LIN {X 0,Y 203.825,Z 341.839,A -85,B 0,C 180,E1 -22082.308,E2 -22082.308} C_VEL
LIN {X 0,Y 207.128,Z 331.94,A -85,B 0,C 180,E1 -22084.047,E2 -22084.047} C_VEL
LIN {X 0,Y 210.227,Z 321.194,A -85,B 0,C 180,E1 -22085.512,E2 -22085.512} C_VEL
LIN {X 0,Y 213.25,Z 308.254,A -85,B 0,C 180,E1 -22086.828,E2 -22086.828} C_VEL
LIN {X 0,Y 215.405,Z 295.863,A -85,B 0,C 180,E1 -22087.718,E2 -22087.718} C_VEL
LIN {X 0,Y 216.743,Z 283.352,A -85,B 0,C 180,E1 -22088.313,E2 -22088.313} C_VEL
LIN {X 0,Y 218.908,Z 244.295,A -85,B 0,C 180,E1 -22089.519,E2 -22089.519} C_VEL
LIN {X 0,Y 217.298,Z 231.269,A -85,B 0,C 180,E1 -22090.465,E2 -22090.465} C_VEL
LIN {X 0,Y 211.83,Z 218.17,A -85,B 0,C 180,E1 -22092.439,E2 -22092.439} C_VEL
LIN {X 0,Y 205.925,Z 205.87,A -85,B 0,C 180,E1 -22094.682,E2 -22094.682} C_VEL
LIN {X 0,Y 200.117,Z 195.617,A -85,B 0,C 180,E1 -22097.023,E2 -22097.023} C_VEL
LIN {X 0,Y 197.007,Z 190.479,A -85,B 0,C 180,E1 -22098.363,E2 -22098.363} C_VEL
LIN {X 0,Y 193.844,Z 185.323,A -85,B 0,C 180,E1 -22099.808,E2 -22099.808} C_VEL
LIN {X 0,Y 190.334,Z 180.05,A -85,B 0,C 180,E1 -22101.501,E2 -22101.501} C_VEL
LIN {X 0,Y 187.044,Z 175.102,A -85,B 0,C 180,E1 -22103.213,E2 -22103.213} C_VEL
LIN {X 0,Y 186.738,Z 174.302,A -85,B 0,C 180,E1 -22103.647,E2 -22103.647} C_VEL
LIN {X 0,Y 185.574,Z 170.368,A -85,B 0,C 180,E1 -22107.043,E2 -22107.043} C_VEL
LIN {X 0,Y 185.551,Z 170.374,A -85,B 0,C 180,E1 -22110.596,E2 -22110.596} C_VEL
LIN {X 0,Y 185.584,Z 170.368,A -85,B 0,C 180,E1 -22115.382,E2 -22115.382} C_VEL
LIN {X 0,Y 185.629,Z 170.346,A -85,B 0,C 180,E1 -22121.18,E2 -22121.18} C_VEL
LIN {X 0,Y 185.7,Z 170.339,A -85,B 0,C 180,E1 -22126.875,E2 -22126.875} C_VEL
LIN {X 0,Y 185.972,Z 170.301,A -85,B 0,C 180,E1 -22131.306,E2 -22131.306} C_VEL
LIN {X 0,Y 186.159,Z 170.279,A -85,B 0,C 180,E1 -22137.837,E2 -22137.837} C_VEL
LIN {X 0,Y 186.378,Z 170.27,A -85,B 0,C 180,E1 -22140,E2 -22140} C_VEL
LIN {X 0,Y 185.881,Z 170.319,A -85,B 0,C 180,E1 -22144.337,E2 -22144.337} C_VEL
LIN {X 0,Y 185.977,Z 170.301,A -85,B 0,C 180,E1 -22148.694,E2 -22148.694} C_VEL
LIN {X 0,Y 185.716,Z 170.338,A -85,B 0,C 180,E1 -22153.124,E2 -22153.124} C_VEL
LIN {X 0,Y 185.655,Z 170.356,A -85,B 0,C 180,E1 -22157.629,E2 -22157.629} C_VEL
LIN {X 0,Y 185.558,Z 170.372,A -85,B 0,C 180,E1 -22162.257,E2 -22162.257} C_VEL
LIN {X 0,Y 185.582,Z 170.355,A -85,B 0,C 180,E1 -22164.646,E2 -22164.646} C_VEL
LIN {X 0,Y 185.549,Z 170.373,A -85,B 0,C 180,E1 -22170.753,E2 -22170.753} C_VEL
LIN {X 0,Y 185.54,Z 170.42,A -85,B 0,C 180,E1 -22171.468,E2 -22171.468} C_VEL
LIN {X 0,Y 186.279,Z 172.794,A -85,B 0,C 180,E1 -22171.967,E2 -22171.967} C_VEL
LIN {X 0,Y 188.238,Z 175.079,A -85,B 0,C 180,E1 -22172.981,E2 -22172.981} C_VEL
LIN {X 0,Y 189.453,Z 176.043,A -85,B 0,C 180,E1 -22173.559,E2 -22173.559} C_VEL
LIN {X 0,Y 191.363,Z 179.22,A -85,B 0,C 180,E1 -22174.539,E2 -22174.539} C_VEL
LIN {X 0,Y 193.288,Z 181.243,A -85,B 0,C 180,E1 -22175.415,E2 -22175.415} C_VEL
LIN {X 0,Y 195.933,Z 184.898,A -85,B 0,C 180,E1 -22176.614,E2 -22176.614} C_VEL
LIN {X 0,Y 202.478,Z 194.218,A -85,B 0,C 180,E1 -22179.344,E2 -22179.344} C_VEL
LIN {X 0,Y 209.512,Z 205.182,A -85,B 0,C 180,E1 -22181.991,E2 -22181.991} C_VEL
LIN {X 0,Y 216.8,Z 218.051,A -85,B 0,C 180,E1 -22184.505,E2 -22184.505} C_VEL
LIN {X 0,Y 219.958,Z 224.99,A -85,B 0,C 180,E1 -22185.571,E2 -22185.571} C_VEL
LIN {X 0,Y 217.34,Z 271.32,A -85,B 0,C 180,E1 -22187.032,E2 -22187.032} C_VEL
LIN {X 0,Y 215.752,Z 284.741,A -85,B 0,C 180,E1 -22187.789,E2 -22187.789} C_VEL
LIN {X 0,Y 213.587,Z 297.23,A -85,B 0,C 180,E1 -22188.844,E2 -22188.844} C_VEL
LIN {X 0,Y 211.086,Z 308.418,A -85,B 0,C 180,E1 -22190.152,E2 -22190.152} C_VEL
LIN {X 0,Y 207.862,Z 319.901,A -85,B 0,C 180,E1 -22191.898,E2 -22191.898} C_VEL
LIN {X 0,Y 204.36,Z 330.28,A -85,B 0,C 180,E1 -22193.917,E2 -22193.917} C_VEL
LIN {X 0,Y 201.13,Z 338.74,A -85,B 0,C 180,E1 -22196.006,E2 -22196.006} C_VEL
LIN {X 0,Y 197.303,Z 347.887,A -85,B 0,C 180,E1 -22198.908,E2 -22198.908} C_VEL
LIN {X 0,Y 193.98,Z 355.197,A -85,B 0,C 180,E1 -22201.899,E2 -22201.899} C_VEL
LIN {X 0,Y 190.993,Z 361.05,A -85,B 0,C 180,E1 -22204.964,E2 -22204.964} C_VEL
LIN {X 0,Y 188.559,Z 365.644,A -85,B 0,C 180,E1 -22208.115,E2 -22208.115} C_VEL
LIN {X 0,Y 187.195,Z 368.068,A -85,B 0,C 180,E1 -22210.25,E2 -22210.25} C_VEL
LIN {X 0,Y 186.035,Z 370.036,A -85,B 0,C 180,E1 -22212.407,E2 -22212.407} C_VEL
LIN {X 0,Y 185.054,Z 371.59,A -85,B 0,C 180,E1 -22214.581,E2 -22214.581} C_VEL
LIN {X 0,Y 184.363,Z 372.721,A -85,B 0,C 180,E1 -22216.776,E2 -22216.776} C_VEL
LIN {X 0,Y 183.555,Z 373.727,A -85,B 0,C 180,E1 -22221.188,E2 -22221.188} C_VEL
LIN {X 0,Y 183.398,Z 373.324,A -85,B 0,C 180,E1 -22225.107,E2 -22225.107} C_VEL
LIN {X 0,Y 183.418,Z 372.318,A -85,B 0,C 180,E1 -22227.802,E2 -22227.802} C_VEL
LIN {X 0,Y 183.588,Z 371.05,A -85,B 0,C 180,E1 -22229.998,E2 -22229.998} C_VEL
LIN {X 0,Y 184.097,Z 368.377,A -85,B 0,C 180,E1 -22233.281,E2 -22233.281} C_VEL
LIN {X 0,Y 185.006,Z 364.704,A -85,B 0,C 180,E1 -22236.542,E2 -22236.542} C_VEL
LIN {X 0,Y 186.412,Z 359.922,A -85,B 0,C 180,E1 -22239.766,E2 -22239.766} C_VEL
LIN {X 0,Y 188.216,Z 353.896,A -85,B 0,C 180,E1 -22242.944,E2 -22242.944} C_VEL
LIN {X 0,Y 190.668,Z 346.391,A -85,B 0,C 180,E1 -22246.046,E2 -22246.046} C_VEL
LIN {X 0,Y 192.991,Z 338.37,A -85,B 0,C 180,E1 -22248.697,E2 -22248.697} C_VEL
LIN {X 0,Y 195.744,Z 328.329,A -85,B 0,C 180,E1 -22251.315,E2 -22251.315} C_VEL
LIN {X 0,Y 198.322,Z 317.738,A -85,B 0,C 180,E1 -22253.493,E2 -22253.493} C_VEL
LIN {X 0,Y 200.493,Z 307.494,A -85,B 0,C 180,E1 -22255.15,E2 -22255.15} C_VEL
LIN {X 0,Y 202.556,Z 295.274,A -85,B 0,C 180,E1 -22256.67,E2 -22256.67} C_VEL
LIN {X 0,Y 204.199,Z 282.413,A -85,B 0,C 180,E1 -22257.823,E2 -22257.823} C_VEL
LIN {X 0,Y 205.326,Z 269.929,A -85,B 0,C 180,E1 -22258.561,E2 -22258.561} C_VEL
LIN {X 0,Y 207.959,Z 212.141,A -85,B 0,C 180,E1 -22260.481,E2 -22260.481} C_VEL
LIN {X 0,Y 202.776,Z 200.79,A -85,B 0,C 180,E1 -22261.935,E2 -22261.935} C_VEL
LIN {X 0,Y 196.04,Z 188.2,A -85,B 0,C 180,E1 -22263.885,E2 -22263.885} C_VEL
LIN {X 0,Y 189.509,Z 177.653,A -85,B 0,C 180,E1 -22265.882,E2 -22265.882} C_VEL
LIN {X 0,Y 187.666,Z 174.56,A -85,B 0,C 180,E1 -22266.486,E2 -22266.486} C_VEL
LIN {X 0,Y 185.986,Z 172.118,A -85,B 0,C 180,E1 -22267.034,E2 -22267.034} C_VEL
LIN {X 0,Y 185.541,Z 170.37,A -85,B 0,C 180,E1 -22267.302,E2 -22267.302} C_VEL
LIN {X 0,Y 185.48,Z 170.377,A -85,B 0,C 180,E1 -22270.727,E2 -22270.727} C_VEL
LIN {X 0,Y 185.455,Z 170.382,A -85,B 0,C 180,E1 -22276.053,E2 -22276.053} C_VEL
LIN {X 0,Y 185.463,Z 170.384,A -85,B 0,C 180,E1 -22279.893,E2 -22279.893} C_VEL
LIN {X 0,Y 185.501,Z 170.372,A -85,B 0,C 180,E1 -22282.709,E2 -22282.709} C_VEL
LIN {X 0,Y 185.536,Z 170.368,A -85,B 0,C 180,E1 -22287.973,E2 -22287.973} C_VEL
LIN {X 0,Y 185.574,Z 170.369,A -85,B 0,C 180,E1 -22290.575,E2 -22290.575} C_VEL
LIN {X 0,Y 185.573,Z 170.371,A -85,B 0,C 180,E1 -22295.38,E2 -22295.38} C_VEL
LIN {X 0,Y 185.625,Z 170.363,A -85,B 0,C 180,E1 -22301.17,E2 -22301.17} C_VEL
LIN {X 0,Y 185.659,Z 170.346,A -85,B 0,C 180,E1 -22304.634,E2 -22304.634} C_VEL
LIN {X 0,Y 185.88,Z 170.324,A -85,B 0,C 180,E1 -22309.419,E2 -22309.419} C_VEL
LIN {X 0,Y 185.919,Z 170.277,A -85,B 0,C 180,E1 -22313.488,E2 -22313.488} C_VEL
LIN {X 0,Y 186.165,Z 170.283,A -85,B 0,C 180,E1 -22317.836,E2 -22317.836} C_VEL
LIN {X 0,Y 186.369,Z 170.269,A -85,B 0,C 180,E1 -22320,E2 -22320} C_VEL
LIN {X 0,Y 185.874,Z 170.331,A -85,B 0,C 180,E1 -22324.337,E2 -22324.337} C_VEL
LIN {X 0,Y 185.963,Z 170.32,A -85,B 0,C 180,E1 -22328.695,E2 -22328.695} C_VEL
LIN {X 0,Y 185.707,Z 170.353,A -85,B 0,C 180,E1 -22333.124,E2 -22333.124} C_VEL
LIN {X 0,Y 185.647,Z 170.362,A -85,B 0,C 180,E1 -22337.629,E2 -22337.629} C_VEL
LIN {X 0,Y 185.565,Z 170.374,A -85,B 0,C 180,E1 -22342.255,E2 -22342.255} C_VEL
LIN {X 0,Y 185.551,Z 170.377,A -85,B 0,C 180,E1 -22347.034,E2 -22347.034} C_VEL
LIN {X 0,Y 185.57,Z 170.372,A -85,B 0,C 180,E1 -22349.495,E2 -22349.495} C_VEL
LIN {X 0,Y 185.492,Z 170.384,A -85,B 0,C 180,E1 -22354.633,E2 -22354.633} C_VEL
LIN {X 0,Y 185.499,Z 170.382,A -85,B 0,C 180,E1 -22357.315,E2 -22357.315} C_VEL
LIN {X 0,Y 185.465,Z 170.385,A -85,B 0,C 180,E1 -22360.726,E2 -22360.726} C_VEL
LIN {X 0,Y 185.477,Z 170.429,A -85,B 0,C 180,E1 -22364.321,E2 -22364.321} C_VEL
LIN {X 0,Y 187.116,Z 176.397,A -85,B 0,C 180,E1 -22367.854,E2 -22367.854} C_VEL
LIN {X 0,Y 189.501,Z 180.912,A -85,B 0,C 180,E1 -22368.662,E2 -22368.662} C_VEL
LIN {X 0,Y 196.299,Z 194.335,A -85,B 0,C 180,E1 -22370.837,E2 -22370.837} C_VEL
LIN {X 0,Y 202.806,Z 209.945,A -85,B 0,C 180,E1 -22372.848,E2 -22372.848} C_VEL
LIN {X 0,Y 204.31,Z 214.184,A -85,B 0,C 180,E1 -22373.315,E2 -22373.315} C_VEL
LIN {X 0,Y 206.787,Z 238.922,A -85,B 0,C 180,E1 -22374.783,E2 -22374.783} C_VEL
LIN {X 0,Y 206.092,Z 255.09,A -85,B 0,C 180,E1 -22375.314,E2 -22375.314} C_VEL
LIN {X 0,Y 205.375,Z 260.94,A -85,B 0,C 180,E1 -22375.412,E2 -22375.412} C_VEL
LIN {X 0,Y 199.61,Z 279.931,A -85,B 0,C 180,E1 -22375.151,E2 -22375.151} C_VEL
LIN {X 0,Y 198.569,Z 285.744,A -85,B 0,C 180,E1 -22375.294,E2 -22375.294} C_VEL
LIN {X 0,Y 197.257,Z 298.93,A -85,B 0,C 180,E1 -22376.098,E2 -22376.098} C_VEL
LIN {X 0,Y 195.306,Z 311.132,A -85,B 0,C 180,E1 -22377.182,E2 -22377.182} C_VEL
LIN {X 0,Y 192.849,Z 323.444,A -85,B 0,C 180,E1 -22378.717,E2 -22378.717} C_VEL
LIN {X 0,Y 190.011,Z 335.076,A -85,B 0,C 180,E1 -22380.657,E2 -22380.657} C_VEL
LIN {X 0,Y 187.159,Z 345.553,A -85,B 0,C 180,E1 -22382.918,E2 -22382.918} C_VEL
LIN {X 0,Y 184.582,Z 354.112,A -85,B 0,C 180,E1 -22385.242,E2 -22385.242} C_VEL
LIN {X 0,Y 182.176,Z 362.221,A -85,B 0,C 180,E1 -22387.993,E2 -22387.993} C_VEL
LIN {X 0,Y 180.295,Z 368.577,A -85,B 0,C 180,E1 -22390.653,E2 -22390.653} C_VEL
LIN {X 0,Y 178.425,Z 375.015,A -85,B 0,C 180,E1 -22393.997,E2 -22393.997} C_VEL
LIN {X 0,Y 177.084,Z 380.127,A -85,B 0,C 180,E1 -22397.394,E2 -22397.394} C_VEL
LIN {X 0,Y 176.4,Z 384.098,A -85,B 0,C 180,E1 -22400.832,E2 -22400.832} C_VEL
LIN {X 0,Y 176.152,Z 386.138,A -85,B 0,C 180,E1 -22403.128,E2 -22403.128} C_VEL
LIN {X 0,Y 176.124,Z 388.127,A -85,B 0,C 180,E1 -22406.022,E2 -22406.022} C_VEL
LIN {X 0,Y 176.323,Z 389.721,A -85,B 0,C 180,E1 -22410.002,E2 -22410.002} C_VEL
LIN {X 0,Y 176.089,Z 390.069,A -85,B 0,C 180,E1 -22413.806,E2 -22413.806} C_VEL
LIN {X 0,Y 176.111,Z 389.563,A -85,B 0,C 180,E1 -22416.878,E2 -22416.878} C_VEL
LIN {X 0,Y 176.388,Z 388.699,A -85,B 0,C 180,E1 -22419.173,E2 -22419.173} C_VEL
LIN {X 0,Y 177.614,Z 385.754,A -85,B 0,C 180,E1 -22423.736,E2 -22423.736} C_VEL
LIN {X 0,Y 179.276,Z 382.422,A -85,B 0,C 180,E1 -22427.1,E2 -22427.1} C_VEL
LIN {X 0,Y 181.534,Z 378.034,A -85,B 0,C 180,E1 -22430.393,E2 -22430.393} C_VEL
LIN {X 0,Y 184.257,Z 372.571,A -85,B 0,C 180,E1 -22433.551,E2 -22433.551} C_VEL
LIN {X 0,Y 187.585,Z 365.547,A -85,B 0,C 180,E1 -22436.719,E2 -22436.719} C_VEL
LIN {X 0,Y 190.915,Z 358.498,A -85,B 0,C 180,E1 -22439.195,E2 -22439.195} C_VEL
LIN {X 0,Y 194.621,Z 350.018,A -85,B 0,C 180,E1 -22441.577,E2 -22441.577} C_VEL
LIN {X 0,Y 198.704,Z 339.558,A -85,B 0,C 180,E1 -22443.855,E2 -22443.855} C_VEL
LIN {X 0,Y 202.628,Z 327.799,A -85,B 0,C 180,E1 -22445.826,E2 -22445.826} C_VEL
LIN {X 0,Y 205.941,Z 316.005,A -85,B 0,C 180,E1 -22447.284,E2 -22447.284} C_VEL
LIN {X 0,Y 208.653,Z 303.751,A -85,B 0,C 180,E1 -22448.393,E2 -22448.393} C_VEL
LIN {X 0,Y 210.672,Z 290.311,A -85,B 0,C 180,E1 -22449.258,E2 -22449.258} C_VEL
LIN {X 0,Y 211.914,Z 275.449,A -85,B 0,C 180,E1 -22449.81,E2 -22449.81} C_VEL
LIN {X 0,Y 213.594,Z 245.006,A -85,B 0,C 180,E1 -22450.76,E2 -22450.76} C_VEL
LIN {X 0,Y 212.13,Z 233.739,A -85,B 0,C 180,E1 -22451.641,E2 -22451.641} C_VEL
LIN {X 0,Y 206.753,Z 220.825,A -85,B 0,C 180,E1 -22453.705,E2 -22453.705} C_VEL
LIN {X 0,Y 201.579,Z 210.06,A -85,B 0,C 180,E1 -22455.79,E2 -22455.79} C_VEL
LIN {X 0,Y 196.244,Z 200.349,A -85,B 0,C 180,E1 -22458.077,E2 -22458.077} C_VEL
LIN {X 0,Y 192.932,Z 194.79,A -85,B 0,C 180,E1 -22459.594,E2 -22459.594} C_VEL
LIN {X 0,Y 190.321,Z 190.463,A -85,B 0,C 180,E1 -22460.862,E2 -22460.862} C_VEL
LIN {X 0,Y 187.146,Z 185.561,A -85,B 0,C 180,E1 -22462.484,E2 -22462.484} C_VEL
LIN {X 0,Y 183.366,Z 179.911,A -85,B 0,C 180,E1 -22464.57,E2 -22464.57} C_VEL
LIN {X 0,Y 180.11,Z 175.501,A -85,B 0,C 180,E1 -22466.505,E2 -22466.505} C_VEL
LIN {X 0,Y 179.416,Z 173.944,A -85,B 0,C 180,E1 -22467.078,E2 -22467.078} C_VEL
LIN {X 0,Y 178.465,Z 171.254,A -85,B 0,C 180,E1 -22469.876,E2 -22469.876} C_VEL
LIN {X 0,Y 178.519,Z 171.247,A -85,B 0,C 180,E1 -22474.89,E2 -22474.89} C_VEL
LIN {X 0,Y 178.609,Z 171.223,A -85,B 0,C 180,E1 -22481.652,E2 -22481.652} C_VEL
LIN {X 0,Y 178.627,Z 171.216,A -85,B 0,C 180,E1 -22486.346,E2 -22486.346} C_VEL
LIN {X 0,Y 178.904,Z 171.182,A -85,B 0,C 180,E1 -22490.96,E2 -22490.96} C_VEL
LIN {X 0,Y 178.819,Z 171.202,A -85,B 0,C 180,E1 -22495.492,E2 -22495.492} C_VEL
LIN {X 0,Y 179.343,Z 171.147,A -85,B 0,C 180,E1 -22500,E2 -22500} C_VEL
LIN {X 0,Y 178.831,Z 171.198,A -85,B 0,C 180,E1 -22504.508,E2 -22504.508} C_VEL
LIN {X 0,Y 178.908,Z 171.181,A -85,B 0,C 180,E1 -22509.041,E2 -22509.041} C_VEL
LIN {X 0,Y 178.642,Z 171.216,A -85,B 0,C 180,E1 -22513.654,E2 -22513.654} C_VEL
LIN {X 0,Y 178.558,Z 171.228,A -85,B 0,C 180,E1 -22519.151,E2 -22519.151} C_VEL
LIN {X 0,Y 178.52,Z 171.236,A -85,B 0,C 180,E1 -22525.111,E2 -22525.111} C_VEL
LIN {X 0,Y 178.461,Z 171.248,A -85,B 0,C 180,E1 -22527.962,E2 -22527.962} C_VEL
LIN {X 0,Y 179.101,Z 173.444,A -85,B 0,C 180,E1 -22528.481,E2 -22528.481} C_VEL
LIN {X 0,Y 181.05,Z 175.861,A -85,B 0,C 180,E1 -22529.68,E2 -22529.68} C_VEL
LIN {X 0,Y 182.667,Z 177.067,A -85,B 0,C 180,E1 -22530.57,E2 -22530.57} C_VEL
LIN {X 0,Y 184.522,Z 180.126,A -85,B 0,C 180,E1 -22531.662,E2 -22531.662} C_VEL
LIN {X 0,Y 186.707,Z 182.45,A -85,B 0,C 180,E1 -22532.798,E2 -22532.798} C_VEL
LIN {X 0,Y 189.354,Z 186.09,A -85,B 0,C 180,E1 -22534.151,E2 -22534.151} C_VEL
LIN {X 0,Y 190.879,Z 188.134,A -85,B 0,C 180,E1 -22534.892,E2 -22534.892} C_VEL
LIN {X 0,Y 194.087,Z 192.584,A -85,B 0,C 180,E1 -22536.382,E2 -22536.382} C_VEL
LIN {X 0,Y 199.121,Z 199.852,A -85,B 0,C 180,E1 -22538.551,E2 -22538.551} C_VEL
LIN {X 0,Y 205.658,Z 210.313,A -85,B 0,C 180,E1 -22541.136,E2 -22541.136} C_VEL
LIN {X 0,Y 212.261,Z 222.203,A -85,B 0,C 180,E1 -22543.537,E2 -22543.537} C_VEL
LIN {X 0,Y 214.588,Z 227.209,A -85,B 0,C 180,E1 -22544.363,E2 -22544.363} C_VEL
LIN {X 0,Y 211.981,Z 271.817,A -85,B 0,C 180,E1 -22545.804,E2 -22545.804} C_VEL
LIN {X 0,Y 210.291,Z 285.444,A -85,B 0,C 180,E1 -22546.589,E2 -22546.589} C_VEL
LIN {X 0,Y 208.265,Z 296.727,A -85,B 0,C 180,E1 -22547.551,E2 -22547.551} C_VEL
LIN {X 0,Y 205.867,Z 307.174,A -85,B 0,C 180,E1 -22548.742,E2 -22548.742} C_VEL
LIN {X 0,Y 202.681,Z 318.438,A -85,B 0,C 180,E1 -22550.418,E2 -22550.418} C_VEL
LIN {X 0,Y 199.044,Z 329.127,A -85,B 0,C 180,E1 -22552.476,E2 -22552.476} C_VEL
LIN {X 0,Y 195.231,Z 338.731,A -85,B 0,C 180,E1 -22554.831,E2 -22554.831} C_VEL
LIN {X 0,Y 191.569,Z 347.247,A -85,B 0,C 180,E1 -22557.543,E2 -22557.543} C_VEL
LIN {X 0,Y 187.706,Z 355.311,A -85,B 0,C 180,E1 -22560.872,E2 -22560.872} C_VEL
LIN {X 0,Y 184.521,Z 361.205,A -85,B 0,C 180,E1 -22564.021,E2 -22564.021} C_VEL
LIN {X 0,Y 181.941,Z 365.834,A -85,B 0,C 180,E1 -22567.275,E2 -22567.275} C_VEL
LIN {X 0,Y 180.477,Z 368.293,A -85,B 0,C 180,E1 -22569.482,E2 -22569.482} C_VEL
LIN {X 0,Y 179.21,Z 370.278,A -85,B 0,C 180,E1 -22571.714,E2 -22571.714} C_VEL
LIN {X 0,Y 178.178,Z 371.846,A -85,B 0,C 180,E1 -22573.97,E2 -22573.97} C_VEL
LIN {X 0,Y 177.392,Z 373.005,A -85,B 0,C 180,E1 -22576.247,E2 -22576.247} C_VEL
LIN {X 0,Y 176.514,Z 374.045,A -85,B 0,C 180,E1 -22580.834,E2 -22580.834} C_VEL
LIN {X 0,Y 176.322,Z 373.61,A -85,B 0,C 180,E1 -22585.194,E2 -22585.194} C_VEL
LIN {X 0,Y 176.317,Z 372.695,A -85,B 0,C 180,E1 -22587.714,E2 -22587.714} C_VEL
LIN {X 0,Y 176.497,Z 371.442,A -85,B 0,C 180,E1 -22589.998,E2 -22589.998} C_VEL
LIN {X 0,Y 177.037,Z 368.8,A -85,B 0,C 180,E1 -22593.412,E2 -22593.412} C_VEL
LIN {X 0,Y 177.983,Z 365.161,A -85,B 0,C 180,E1 -22596.801,E2 -22596.801} C_VEL
LIN {X 0,Y 179.447,Z 360.415,A -85,B 0,C 180,E1 -22600.149,E2 -22600.149} C_VEL
LIN {X 0,Y 181.346,Z 354.427,A -85,B 0,C 180,E1 -22603.444,E2 -22603.444} C_VEL
LIN {X 0,Y 183.897,Z 346.967,A -85,B 0,C 180,E1 -22606.654,E2 -22606.654} C_VEL
LIN {X 0,Y 186.489,Z 338.386,A -85,B 0,C 180,E1 -22609.584,E2 -22609.584} C_VEL
LIN {X 0,Y 189.467,Z 327.992,A -85,B 0,C 180,E1 -22612.344,E2 -22612.344} C_VEL
LIN {X 0,Y 192.209,Z 317.256,A -85,B 0,C 180,E1 -22614.575,E2 -22614.575} C_VEL
LIN {X 0,Y 194.489,Z 306.782,A -85,B 0,C 180,E1 -22616.271,E2 -22616.271} C_VEL
LIN {X 0,Y 196.643,Z 294.2,A -85,B 0,C 180,E1 -22617.828,E2 -22617.828} C_VEL
LIN {X 0,Y 198.273,Z 281.609,A -85,B 0,C 180,E1 -22618.948,E2 -22618.948} C_VEL
LIN {X 0,Y 199.398,Z 268.524,A -85,B 0,C 180,E1 -22619.693,E2 -22619.693} C_VEL
LIN {X 0,Y 202.004,Z 214.055,A -85,B 0,C 180,E1 -22621.525,E2 -22621.525} C_VEL
LIN {X 0,Y 195.871,Z 201.044,A -85,B 0,C 180,E1 -22623.347,E2 -22623.347} C_VEL
LIN {X 0,Y 189.283,Z 189.159,A -85,B 0,C 180,E1 -22625.389,E2 -22625.389} C_VEL
LIN {X 0,Y 183.018,Z 179.167,A -85,B 0,C 180,E1 -22627.461,E2 -22627.461} C_VEL
LIN {X 0,Y 180.81,Z 175.727,A -85,B 0,C 180,E1 -22628.238,E2 -22628.238} C_VEL
LIN {X 0,Y 179.093,Z 173.472,A -85,B 0,C 180,E1 -22628.839,E2 -22628.839} C_VEL
LIN {X 0,Y 178.416,Z 171.257,A -85,B 0,C 180,E1 -22629.207,E2 -22629.207} C_VEL
LIN {X 0,Y 178.398,Z 171.261,A -85,B 0,C 180,E1 -22632.042,E2 -22632.042} C_VEL
LIN {X 0,Y 178.389,Z 171.264,A -85,B 0,C 180,E1 -22635.162,E2 -22635.162} C_VEL
LIN {X 0,Y 178.398,Z 171.259,A -85,B 0,C 180,E1 -22638.457,E2 -22638.457} C_VEL
LIN {X 0,Y 178.417,Z 171.26,A -85,B 0,C 180,E1 -22643.781,E2 -22643.781} C_VEL
LIN {X 0,Y 178.479,Z 171.246,A -85,B 0,C 180,E1 -22646.545,E2 -22646.545} C_VEL
LIN {X 0,Y 178.515,Z 171.25,A -85,B 0,C 180,E1 -22650.006,E2 -22650.006} C_VEL
LIN {X 0,Y 178.513,Z 171.248,A -85,B 0,C 180,E1 -22654.885,E2 -22654.885} C_VEL
LIN {X 0,Y 178.582,Z 171.239,A -85,B 0,C 180,E1 -22660.814,E2 -22660.814} C_VEL
LIN {X 0,Y 178.634,Z 171.23,A -85,B 0,C 180,E1 -22666.346,E2 -22666.346} C_VEL
LIN {X 0,Y 178.895,Z 171.178,A -85,B 0,C 180,E1 -22670.959,E2 -22670.959} C_VEL
LIN {X 0,Y 179.112,Z 171.159,A -85,B 0,C 180,E1 -22677.751,E2 -22677.751} C_VEL
LIN {X 0,Y 179.335,Z 171.146,A -85,B 0,C 180,E1 -22680,E2 -22680} C_VEL
LIN {X 0,Y 178.823,Z 171.209,A -85,B 0,C 180,E1 -22684.508,E2 -22684.508} C_VEL
LIN {X 0,Y 178.894,Z 171.202,A -85,B 0,C 180,E1 -22689.041,E2 -22689.041} C_VEL
LIN {X 0,Y 178.634,Z 171.236,A -85,B 0,C 180,E1 -22693.654,E2 -22693.654} C_VEL
LIN {X 0,Y 178.582,Z 171.243,A -85,B 0,C 180,E1 -22699.186,E2 -22699.186} C_VEL
LIN {X 0,Y 178.512,Z 171.249,A -85,B 0,C 180,E1 -22705.115,E2 -22705.115} C_VEL
LIN {X 0,Y 178.514,Z 171.253,A -85,B 0,C 180,E1 -22709.994,E2 -22709.994} C_VEL
LIN {X 0,Y 178.477,Z 171.259,A -85,B 0,C 180,E1 -22714.22,E2 -22714.22} C_VEL
LIN {X 0,Y 178.389,Z 171.268,A -85,B 0,C 180,E1 -22719.076,E2 -22719.076} C_VEL
LIN {X 0,Y 178.437,Z 171.439,A -85,B 0,C 180,E1 -22722.99,E2 -22722.99} C_VEL
LIN {X 0,Y 179.68,Z 175.934,A -85,B 0,C 180,E1 -22725.847,E2 -22725.847} C_VEL
LIN {X 0,Y 182.122,Z 180.378,A -85,B 0,C 180,E1 -22726.75,E2 -22726.75} C_VEL
LIN {X 0,Y 187.929,Z 191.354,A -85,B 0,C 180,E1 -22728.779,E2 -22728.779} C_VEL
LIN {X 0,Y 192.702,Z 201.504,A -85,B 0,C 180,E1 -22730.368,E2 -22730.368} C_VEL
LIN {X 0,Y 198.548,Z 216.235,A -85,B 0,C 180,E1 -22732.271,E2 -22732.271} C_VEL
LIN {X 0,Y 200.811,Z 239.813,A -85,B 0,C 180,E1 -22733.723,E2 -22733.723} C_VEL
LIN {X 0,Y 198.569,Z 285.744,A -85,B 0,C 180,E1 -22735.294,E2 -22735.294} C_VEL
LIN {X 0,Y 197.902,Z 289.61,A -85,B 0,C 180,E1 -22735.426,E2 -22735.426} C_VEL
LIN {X 0,Y 195.365,Z 297.109,A -85,B 0,C 180,E1 -22735.586,E2 -22735.586} C_VEL
LIN {X 0,Y 190.602,Z 307.98,A -85,B 0,C 180,E1 -22735.95,E2 -22735.95} C_VEL
LIN {X 0,Y 188.792,Z 313.448,A -85,B 0,C 180,E1 -22736.398,E2 -22736.398} C_VEL
LIN {X 0,Y 188.386,Z 315.225,A -85,B 0,C 180,E1 -22736.603,E2 -22736.603} C_VEL
LIN {X 0,Y 185.619,Z 327.365,A -85,B 0,C 180,E1 -22738.312,E2 -22738.312} C_VEL
LIN {X 0,Y 182.808,Z 338.119,A -85,B 0,C 180,E1 -22740.335,E2 -22740.335} C_VEL
LIN {X 0,Y 179.842,Z 347.915,A -85,B 0,C 180,E1 -22742.669,E2 -22742.669} C_VEL
LIN {X 0,Y 177.099,Z 356.849,A -85,B 0,C 180,E1 -22745.377,E2 -22745.377} C_VEL
LIN {X 0,Y 174.93,Z 364.028,A -85,B 0,C 180,E1 -22748.094,E2 -22748.094} C_VEL
LIN {X 0,Y 172.56,Z 371.486,A -85,B 0,C 180,E1 -22751.603,E2 -22751.603} C_VEL
LIN {X 0,Y 170.994,Z 376.375,A -85,B 0,C 180,E1 -22754.507,E2 -22754.507} C_VEL
LIN {X 0,Y 169.807,Z 381.133,A -85,B 0,C 180,E1 -22758.059,E2 -22758.059} C_VEL
LIN {X 0,Y 169.196,Z 384.768,A -85,B 0,C 180,E1 -22761.643,E2 -22761.643} C_VEL
LIN {X 0,Y 169.03,Z 387.957,A -85,B 0,C 180,E1 -22766.268,E2 -22766.268} C_VEL
LIN {X 0,Y 169.24,Z 389.379,A -85,B 0,C 180,E1 -22770.002,E2 -22770.002} C_VEL
LIN {X 0,Y 168.998,Z 389.78,A -85,B 0,C 180,E1 -22773.562,E2 -22773.562} C_VEL
LIN {X 0,Y 169.032,Z 389.257,A -85,B 0,C 180,E1 -22777.167,E2 -22777.167} C_VEL
LIN {X 0,Y 169.353,Z 388.418,A -85,B 0,C 180,E1 -22779.557,E2 -22779.557} C_VEL
LIN {X 0,Y 169.913,Z 387.159,A -85,B 0,C 180,E1 -22781.938,E2 -22781.938} C_VEL
LIN {X 0,Y 171.185,Z 384.514,A -85,B 0,C 180,E1 -22785.479,E2 -22785.479} C_VEL
LIN {X 0,Y 173.237,Z 380.876,A -85,B 0,C 180,E1 -22788.94,E2 -22788.94} C_VEL
LIN {X 0,Y 175.858,Z 376.142,A -85,B 0,C 180,E1 -22792.314,E2 -22792.314} C_VEL
LIN {X 0,Y 179.453,Z 369.046,A -85,B 0,C 180,E1 -22796.143,E2 -22796.143} C_VEL
LIN {X 0,Y 183.287,Z 361.384,A -85,B 0,C 180,E1 -22799.269,E2 -22799.269} C_VEL
LIN {X 0,Y 187.829,Z 351.778,A -85,B 0,C 180,E1 -22802.223,E2 -22802.223} C_VEL
LIN {X 0,Y 191.986,Z 341.885,A -85,B 0,C 180,E1 -22804.571,E2 -22804.571} C_VEL
LIN {X 0,Y 195.565,Z 332.173,A -85,B 0,C 180,E1 -22806.369,E2 -22806.369} C_VEL
LIN {X 0,Y 198.889,Z 321.681,A -85,B 0,C 180,E1 -22807.879,E2 -22807.879} C_VEL
LIN {X 0,Y 202.105,Z 309.061,A -85,B 0,C 180,E1 -22809.233,E2 -22809.233} C_VEL
LIN {X 0,Y 204.67,Z 295.705,A -85,B 0,C 180,E1 -22810.241,E2 -22810.241} C_VEL
LIN {X 0,Y 206.14,Z 283.137,A -85,B 0,C 180,E1 -22810.866,E2 -22810.866} C_VEL
LIN {X 0,Y 208.409,Z 246.562,A -85,B 0,C 180,E1 -22812.019,E2 -22812.019} C_VEL
LIN {X 0,Y 207.259,Z 236.916,A -85,B 0,C 180,E1 -22812.787,E2 -22812.787} C_VEL
LIN {X 0,Y 202.288,Z 224.696,A -85,B 0,C 180,E1 -22814.819,E2 -22814.819} C_VEL
LIN {X 0,Y 197.31,Z 214.161,A -85,B 0,C 180,E1 -22816.952,E2 -22816.952} C_VEL
LIN {X 0,Y 192.544,Z 205.245,A -85,B 0,C 180,E1 -22819.126,E2 -22819.126} C_VEL
LIN {X 0,Y 187.171,Z 195.994,A -85,B 0,C 180,E1 -22821.803,E2 -22821.803} C_VEL
LIN {X 0,Y 183.761,Z 190.707,A -85,B 0,C 180,E1 -22823.642,E2 -22823.642} C_VEL
LIN {X 0,Y 180.501,Z 185.654,A -85,B 0,C 180,E1 -22825.556,E2 -22825.556} C_VEL
LIN {X 0,Y 177.317,Z 181.146,A -85,B 0,C 180,E1 -22827.567,E2 -22827.567} C_VEL
LIN {X 0,Y 176.469,Z 179.766,A -85,B 0,C 180,E1 -22828.151,E2 -22828.151} C_VEL
LIN {X 0,Y 172.056,Z 174.359,A -85,B 0,C 180,E1 -22831.318,E2 -22831.318} C_VEL
LIN {X 0,Y 171.663,Z 173.261,A -85,B 0,C 180,E1 -22831.746,E2 -22831.746} C_VEL
LIN {X 0,Y 171.393,Z 172.135,A -85,B 0,C 180,E1 -22833.189,E2 -22833.189} C_VEL
LIN {X 0,Y 171.44,Z 172.128,A -85,B 0,C 180,E1 -22835.799,E2 -22835.799} C_VEL
LIN {X 0,Y 171.511,Z 172.103,A -85,B 0,C 180,E1 -22840.864,E2 -22840.864} C_VEL
LIN {X 0,Y 171.543,Z 172.098,A -85,B 0,C 180,E1 -22845.77,E2 -22845.77} C_VEL
LIN {X 0,Y 171.844,Z 172.063,A -85,B 0,C 180,E1 -22850.585,E2 -22850.585} C_VEL
LIN {X 0,Y 171.77,Z 172.081,A -85,B 0,C 180,E1 -22855.306,E2 -22855.306} C_VEL
LIN {X 0,Y 172.307,Z 172.023,A -85,B 0,C 180,E1 -22860,E2 -22860} C_VEL
LIN {X 0,Y 171.781,Z 172.078,A -85,B 0,C 180,E1 -22864.694,E2 -22864.694} C_VEL
LIN {X 0,Y 171.847,Z 172.062,A -85,B 0,C 180,E1 -22869.415,E2 -22869.415} C_VEL
LIN {X 0,Y 171.557,Z 172.097,A -85,B 0,C 180,E1 -22874.229,E2 -22874.229} C_VEL
LIN {X 0,Y 171.484,Z 172.108,A -85,B 0,C 180,E1 -22879.499,E2 -22879.499} C_VEL
LIN {X 0,Y 171.436,Z 172.117,A -85,B 0,C 180,E1 -22883.72,E2 -22883.72} C_VEL
LIN {X 0,Y 172.179,Z 174.498,A -85,B 0,C 180,E1 -22884.452,E2 -22884.452} C_VEL
LIN {X 0,Y 174.332,Z 177.012,A -85,B 0,C 180,E1 -22886.041,E2 -22886.041} C_VEL
LIN {X 0,Y 175.958,Z 178.166,A -85,B 0,C 180,E1 -22887.103,E2 -22887.103} C_VEL
LIN {X 0,Y 177.721,Z 181.147,A -85,B 0,C 180,E1 -22888.33,E2 -22888.33} C_VEL
LIN {X 0,Y 180.141,Z 183.519,A -85,B 0,C 180,E1 -22889.782,E2 -22889.782} C_VEL
LIN {X 0,Y 182.625,Z 187.014,A -85,B 0,C 180,E1 -22891.25,E2 -22891.25} C_VEL
LIN {X 0,Y 183.988,Z 188.588,A -85,B 0,C 180,E1 -22891.993,E2 -22891.993} C_VEL
LIN {X 0,Y 186.846,Z 192.383,A -85,B 0,C 180,E1 -22893.504,E2 -22893.504} C_VEL
LIN {X 0,Y 191.527,Z 199.152,A -85,B 0,C 180,E1 -22895.808,E2 -22895.808} C_VEL
LIN {X 0,Y 196.002,Z 205.831,A -85,B 0,C 180,E1 -22897.82,E2 -22897.82} C_VEL
LIN {X 0,Y 201.943,Z 215.539,A -85,B 0,C 180,E1 -22900.282,E2 -22900.282} C_VEL
LIN {X 0,Y 208.384,Z 227.47,A -85,B 0,C 180,E1 -22902.746,E2 -22902.746} C_VEL
LIN {X 0,Y 209.391,Z 229.675,A -85,B 0,C 180,E1 -22903.124,E2 -22903.124} C_VEL
LIN {X 0,Y 206.81,Z 271.373,A -85,B 0,C 180,E1 -22904.466,E2 -22904.466} C_VEL
LIN {X 0,Y 205.154,Z 284.621,A -85,B 0,C 180,E1 -22905.216,E2 -22905.216} C_VEL
LIN {X 0,Y 202.847,Z 297.237,A -85,B 0,C 180,E1 -22906.292,E2 -22906.292} C_VEL
LIN {X 0,Y 200.201,Z 308.23,A -85,B 0,C 180,E1 -22907.578,E2 -22907.578} C_VEL
LIN {X 0,Y 196.802,Z 319.575,A -85,B 0,C 180,E1 -22909.326,E2 -22909.326} C_VEL
LIN {X 0,Y 193.002,Z 330.122,A -85,B 0,C 180,E1 -22911.419,E2 -22911.419} C_VEL
LIN {X 0,Y 189.405,Z 338.721,A -85,B 0,C 180,E1 -22913.579,E2 -22913.579} C_VEL
LIN {X 0,Y 185.59,Z 347.216,A -85,B 0,C 180,E1 -22916.313,E2 -22916.313} C_VEL
LIN {X 0,Y 182.121,Z 354.311,A -85,B 0,C 180,E1 -22919.247,E2 -22919.247} C_VEL
LIN {X 0,Y 179.162,Z 359.554,A -85,B 0,C 180,E1 -22921.917,E2 -22921.917} C_VEL
LIN {X 0,Y 176.192,Z 364.611,A -85,B 0,C 180,E1 -22925.238,E2 -22925.238} C_VEL
LIN {X 0,Y 173.757,Z 368.519,A -85,B 0,C 180,E1 -22928.65,E2 -22928.65} C_VEL
LIN {X 0,Y 172.417,Z 370.52,A -85,B 0,C 180,E1 -22930.966,E2 -22930.966} C_VEL
LIN {X 0,Y 171.325,Z 372.103,A -85,B 0,C 180,E1 -22933.311,E2 -22933.311} C_VEL
LIN {X 0,Y 170.442,Z 373.284,A -85,B 0,C 180,E1 -22935.674,E2 -22935.674} C_VEL
LIN {X 0,Y 169.861,Z 374.021,A -85,B 0,C 180,E1 -22938.059,E2 -22938.059} C_VEL
LIN {X 0,Y 169.263,Z 374.324,A -85,B 0,C 180,E1 -22942.842,E2 -22942.842} C_VEL
LIN {X 0,Y 169.215,Z 373.86,A -85,B 0,C 180,E1 -22945.417,E2 -22945.417} C_VEL
LIN {X 0,Y 169.408,Z 371.834,A -85,B 0,C 180,E1 -22949.998,E2 -22949.998} C_VEL
LIN {X 0,Y 169.979,Z 369.222,A -85,B 0,C 180,E1 -22953.554,E2 -22953.554} C_VEL
LIN {X 0,Y 170.966,Z 365.617,A -85,B 0,C 180,E1 -22957.082,E2 -22957.082} C_VEL
LIN {X 0,Y 172.493,Z 360.907,A -85,B 0,C 180,E1 -22960.562,E2 -22960.562} C_VEL
LIN {X 0,Y 174.903,Z 353.849,A -85,B 0,C 180,E1 -22964.542,E2 -22964.542} C_VEL
LIN {X 0,Y 177.609,Z 346.151,A -85,B 0,C 180,E1 -22967.856,E2 -22967.856} C_VEL
LIN {X 0,Y 180.079,Z 338.301,A -85,B 0,C 180,E1 -22970.561,E2 -22970.561} C_VEL
LIN {X 0,Y 183.267,Z 327.654,A -85,B 0,C 180,E1 -22973.442,E2 -22973.442} C_VEL
LIN {X 0,Y 186.12,Z 316.726,A -85,B 0,C 180,E1 -22975.735,E2 -22975.735} C_VEL
LIN {X 0,Y 188.56,Z 306.012,A -85,B 0,C 180,E1 -22977.465,E2 -22977.465} C_VEL
LIN {X 0,Y 190.617,Z 294.249,A -85,B 0,C 180,E1 -22978.939,E2 -22978.939} C_VEL
LIN {X 0,Y 192.33,Z 281.554,A -85,B 0,C 180,E1 -22980.083,E2 -22980.083} C_VEL
LIN {X 0,Y 193.505,Z 268.264,A -85,B 0,C 180,E1 -22980.836,E2 -22980.836} C_VEL
LIN {X 0,Y 196.11,Z 216.113,A -85,B 0,C 180,E1 -22982.627,E2 -22982.627} C_VEL
LIN {X 0,Y 189.768,Z 202.822,A -85,B 0,C 180,E1 -22984.631,E2 -22984.631} C_VEL
LIN {X 0,Y 183.404,Z 191.508,A -85,B 0,C 180,E1 -22986.74,E2 -22986.74} C_VEL
LIN {X 0,Y 176.69,Z 180.891,A -85,B 0,C 180,E1 -22989.14,E2 -22989.14} C_VEL
LIN {X 0,Y 174.562,Z 177.719,A -85,B 0,C 180,E1 -22989.949,E2 -22989.949} C_VEL
LIN {X 0,Y 173.542,Z 176.345,A -85,B 0,C 180,E1 -22990.339,E2 -22990.339} C_VEL
LIN {X 0,Y 171.902,Z 174.048,A -85,B 0,C 180,E1 -22990.987,E2 -22990.987} C_VEL
LIN {X 0,Y 171.391,Z 172.131,A -85,B 0,C 180,E1 -22991.297,E2 -22991.297} C_VEL
LIN {X 0,Y 171.316,Z 172.144,A -85,B 0,C 180,E1 -22995.781,E2 -22995.781} C_VEL
LIN {X 0,Y 171.352,Z 172.135,A -85,B 0,C 180,E1 -23001.191,E2 -23001.191} C_VEL
LIN {X 0,Y 171.392,Z 172.137,A -85,B 0,C 180,E1 -23005.091,E2 -23005.091} C_VEL
LIN {X 0,Y 171.441,Z 172.13,A -85,B 0,C 180,E1 -23010.532,E2 -23010.532} C_VEL
LIN {X 0,Y 171.436,Z 172.131,A -85,B 0,C 180,E1 -23015.798,E2 -23015.798} C_VEL
LIN {X 0,Y 171.538,Z 172.116,A -85,B 0,C 180,E1 -23020.866,E2 -23020.866} C_VEL
LIN {X 0,Y 171.549,Z 172.108,A -85,B 0,C 180,E1 -23025.77,E2 -23025.77} C_VEL
LIN {X 0,Y 171.834,Z 172.06,A -85,B 0,C 180,E1 -23030.584,E2 -23030.584} C_VEL
LIN {X 0,Y 171.769,Z 172.04,A -85,B 0,C 180,E1 -23035.306,E2 -23035.306} C_VEL
LIN {X 0,Y 172.299,Z 172.022,A -85,B 0,C 180,E1 -23040,E2 -23040} C_VEL
LIN {X 0,Y 171.773,Z 172.088,A -85,B 0,C 180,E1 -23044.693,E2 -23044.693} C_VEL
LIN {X 0,Y 171.833,Z 172.083,A -85,B 0,C 180,E1 -23049.416,E2 -23049.416} C_VEL
LIN {X 0,Y 171.549,Z 172.119,A -85,B 0,C 180,E1 -23054.229,E2 -23054.229} C_VEL
LIN {X 0,Y 171.507,Z 172.124,A -85,B 0,C 180,E1 -23059.534,E2 -23059.534} C_VEL
LIN {X 0,Y 171.451,Z 172.131,A -85,B 0,C 180,E1 -23065.61,E2 -23065.61} C_VEL
LIN {X 0,Y 171.433,Z 172.137,A -85,B 0,C 180,E1 -23070.587,E2 -23070.587} C_VEL
LIN {X 0,Y 171.386,Z 172.141,A -85,B 0,C 180,E1 -23075.036,E2 -23075.036} C_VEL
LIN {X 0,Y 171.351,Z 172.145,A -85,B 0,C 180,E1 -23078.809,E2 -23078.809} C_VEL
LIN {X 0,Y 171.346,Z 172.148,A -85,B 0,C 180,E1 -23081.317,E2 -23081.317} C_VEL
LIN {X 0,Y 172.347,Z 175.674,A -85,B 0,C 180,E1 -23083.638,E2 -23083.638} C_VEL
LIN {X 0,Y 175.178,Z 180.513,A -85,B 0,C 180,E1 -23084.781,E2 -23084.781} C_VEL
LIN {X 0,Y 181.759,Z 192.718,A -85,B 0,C 180,E1 -23087.279,E2 -23087.279} C_VEL
LIN {X 0,Y 186.847,Z 203.451,A -85,B 0,C 180,E1 -23089.097,E2 -23089.097} C_VEL
LIN {X 0,Y 192.527,Z 217.674,A -85,B 0,C 180,E1 -23091.067,E2 -23091.067} C_VEL
LIN {X 0,Y 193.093,Z 220.458,A -85,B 0,C 180,E1 -23091.316,E2 -23091.316} C_VEL
LIN {X 0,Y 194.919,Z 240.316,A -85,B 0,C 180,E1 -23092.584,E2 -23092.584} C_VEL
LIN {X 0,Y 192.568,Z 285.988,A -85,B 0,C 180,E1 -23094.19,E2 -23094.19} C_VEL
LIN {X 0,Y 191.185,Z 299.157,A -85,B 0,C 180,E1 -23095.027,E2 -23095.027} C_VEL
LIN {X 0,Y 189.162,Z 311.217,A -85,B 0,C 180,E1 -23096.134,E2 -23096.134} C_VEL
LIN {X 0,Y 188.386,Z 315.225,A -85,B 0,C 180,E1 -23096.603,E2 -23096.603} C_VEL
LIN {X 0,Y 187.06,Z 318.828,A -85,B 0,C 180,E1 -23096.953,E2 -23096.953} C_VEL
LIN {X 0,Y 183.254,Z 324.333,A -85,B 0,C 180,E1 -23097.291,E2 -23097.291} C_VEL
LIN {X 0,Y 179.357,Z 329.666,A -85,B 0,C 180,E1 -23097.746,E2 -23097.746} C_VEL
LIN {X 0,Y 177.902,Z 332.971,A -85,B 0,C 180,E1 -23098.281,E2 -23098.281} C_VEL
LIN {X 0,Y 174.533,Z 344.207,A -85,B 0,C 180,E1 -23100.778,E2 -23100.778} C_VEL
LIN {X 0,Y 171.701,Z 352.884,A -85,B 0,C 180,E1 -23103.243,E2 -23103.243} C_VEL
LIN {X 0,Y 168.997,Z 361.144,A -85,B 0,C 180,E1 -23106.192,E2 -23106.192} C_VEL
LIN {X 0,Y 166.926,Z 367.532,A -85,B 0,C 180,E1 -23109.033,E2 -23109.033} C_VEL
LIN {X 0,Y 164.744,Z 374.063,A -85,B 0,C 180,E1 -23112.628,E2 -23112.628} C_VEL
LIN {X 0,Y 163.155,Z 379.244,A -85,B 0,C 180,E1 -23116.298,E2 -23116.298} C_VEL
LIN {X 0,Y 162.331,Z 383.275,A -85,B 0,C 180,E1 -23120.03,E2 -23120.03} C_VEL
LIN {X 0,Y 162.018,Z 385.345,A -85,B 0,C 180,E1 -23122.525,E2 -23122.525} C_VEL
LIN {X 0,Y 161.959,Z 387.735,A -85,B 0,C 180,E1 -23126.425,E2 -23126.425} C_VEL
LIN {X 0,Y 162.158,Z 389.037,A -85,B 0,C 180,E1 -23130.002,E2 -23130.002} C_VEL
LIN {X 0,Y 161.913,Z 389.437,A -85,B 0,C 180,E1 -23133.303,E2 -23133.303} C_VEL
LIN {X 0,Y 161.963,Z 388.951,A -85,B 0,C 180,E1 -23137.482,E2 -23137.482} C_VEL
LIN {X 0,Y 162.339,Z 388.138,A -85,B 0,C 180,E1 -23139.974,E2 -23139.974} C_VEL
LIN {X 0,Y 163.759,Z 385.245,A -85,B 0,C 180,E1 -23144.924,E2 -23144.924} C_VEL
LIN {X 0,Y 165.709,Z 381.971,A -85,B 0,C 180,E1 -23148.549,E2 -23148.549} C_VEL
LIN {X 0,Y 168.26,Z 377.644,A -85,B 0,C 180,E1 -23152.083,E2 -23152.083} C_VEL
LIN {X 0,Y 171.928,Z 371.097,A -85,B 0,C 180,E1 -23156.09,E2 -23156.09} C_VEL
LIN {X 0,Y 175.667,Z 364.006,A -85,B 0,C 180,E1 -23159.349,E2 -23159.349} C_VEL
LIN {X 0,Y 180.209,Z 355.157,A -85,B 0,C 180,E1 -23162.43,E2 -23162.43} C_VEL
LIN {X 0,Y 184.371,Z 346.102,A -85,B 0,C 180,E1 -23164.876,E2 -23164.876} C_VEL
LIN {X 0,Y 188.472,Z 336.134,A -85,B 0,C 180,E1 -23166.964,E2 -23166.964} C_VEL
LIN {X 0,Y 192.333,Z 325.068,A -85,B 0,C 180,E1 -23168.74,E2 -23168.74} C_VEL
LIN {X 0,Y 195.91,Z 312.675,A -85,B 0,C 180,E1 -23170.222,E2 -23170.222} C_VEL
LIN {X 0,Y 198.529,Z 300.894,A -85,B 0,C 180,E1 -23171.251,E2 -23171.251} C_VEL
LIN {X 0,Y 200.509,Z 287.662,A -85,B 0,C 180,E1 -23172.045,E2 -23172.045} C_VEL
LIN {X 0,Y 202.015,Z 268.304,A -85,B 0,C 180,E1 -23172.721,E2 -23172.721} C_VEL
LIN {X 0,Y 203.313,Z 247.554,A -85,B 0,C 180,E1 -23173.374,E2 -23173.374} C_VEL
LIN {X 0,Y 202.464,Z 240.025,A -85,B 0,C 180,E1 -23173.993,E2 -23173.993} C_VEL
LIN {X 0,Y 197.109,Z 226.645,A -85,B 0,C 180,E1 -23176.344,E2 -23176.344} C_VEL
LIN {X 0,Y 191.821,Z 215.61,A -85,B 0,C 180,E1 -23178.789,E2 -23178.789} C_VEL
LIN {X 0,Y 186.296,Z 205.491,A -85,B 0,C 180,E1 -23181.563,E2 -23181.563} C_VEL
LIN {X 0,Y 183.227,Z 200.262,A -85,B 0,C 180,E1 -23183.237,E2 -23183.237} C_VEL
LIN {X 0,Y 179.892,Z 194.93,A -85,B 0,C 180,E1 -23185.186,E2 -23185.186} C_VEL
LIN {X 0,Y 177.723,Z 191.424,A -85,B 0,C 180,E1 -23186.554,E2 -23186.554} C_VEL
LIN {X 0,Y 174.52,Z 186.637,A -85,B 0,C 180,E1 -23188.715,E2 -23188.715} C_VEL
LIN {X 0,Y 169.681,Z 180.237,A -85,B 0,C 180,E1 -23192.395,E2 -23192.395} C_VEL
LIN {X 0,Y 168.761,Z 178.824,A -85,B 0,C 180,E1 -23193.199,E2 -23193.199} C_VEL
LIN {X 0,Y 165.833,Z 176.485,A -85,B 0,C 180,E1 -23195.76,E2 -23195.76} C_VEL
LIN {X 0,Y 164.574,Z 174.11,A -85,B 0,C 180,E1 -23197.149,E2 -23197.149} C_VEL
LIN {X 0,Y 164.359,Z 173.011,A -85,B 0,C 180,E1 -23197.532,E2 -23197.532} C_VEL
LIN {X 0,Y 164.431,Z 172.998,A -85,B 0,C 180,E1 -23202.591,E2 -23202.591} C_VEL
LIN {X 0,Y 164.704,Z 172.969,A -85,B 0,C 180,E1 -23208.945,E2 -23208.945} C_VEL
LIN {X 0,Y 164.818,Z 172.939,A -85,B 0,C 180,E1 -23212.651,E2 -23212.651} C_VEL
LIN {X 0,Y 165.272,Z 172.899,A -85,B 0,C 180,E1 -23220,E2 -23220} C_VEL
LIN {X 0,Y 164.822,Z 172.941,A -85,B 0,C 180,E1 -23227.35,E2 -23227.35} C_VEL
LIN {X 0,Y 164.706,Z 172.967,A -85,B 0,C 180,E1 -23231.058,E2 -23231.058} C_VEL
LIN {X 0,Y 164.44,Z 172.999,A -85,B 0,C 180,E1 -23237.408,E2 -23237.408} C_VEL
LIN {X 0,Y 164.457,Z 173.05,A -85,B 0,C 180,E1 -23238.291,E2 -23238.291} C_VEL
LIN {X 0,Y 165.221,Z 175.413,A -85,B 0,C 180,E1 -23239.263,E2 -23239.263} C_VEL
LIN {X 0,Y 166.954,Z 177.642,A -85,B 0,C 180,E1 -23240.966,E2 -23240.966} C_VEL
LIN {X 0,Y 169.223,Z 179.025,A -85,B 0,C 180,E1 -23242.834,E2 -23242.834} C_VEL
LIN {X 0,Y 170.892,Z 182.031,A -85,B 0,C 180,E1 -23244.284,E2 -23244.284} C_VEL
LIN {X 0,Y 173.631,Z 184.618,A -85,B 0,C 180,E1 -23246.261,E2 -23246.261} C_VEL
LIN {X 0,Y 175.808,Z 187.837,A -85,B 0,C 180,E1 -23247.798,E2 -23247.798} C_VEL
LIN {X 0,Y 177.676,Z 189.848,A -85,B 0,C 180,E1 -23248.977,E2 -23248.977} C_VEL
LIN {X 0,Y 180.555,Z 193.634,A -85,B 0,C 180,E1 -23250.723,E2 -23250.723} C_VEL
LIN {X 0,Y 185.684,Z 200.845,A -85,B 0,C 180,E1 -23253.555,E2 -23253.555} C_VEL
LIN {X 0,Y 191.733,Z 209.797,A -85,B 0,C 180,E1 -23256.514,E2 -23256.514} C_VEL
LIN {X 0,Y 198.023,Z 220.383,A -85,B 0,C 180,E1 -23259.294,E2 -23259.294} C_VEL
LIN {X 0,Y 204.022,Z 231.745,A -85,B 0,C 180,E1 -23261.723,E2 -23261.723} C_VEL
LIN {X 0,Y 204.203,Z 232.11,A -85,B 0,C 180,E1 -23261.794,E2 -23261.794} C_VEL
LIN {X 0,Y 201.616,Z 272.232,A -85,B 0,C 180,E1 -23263.121,E2 -23263.121} C_VEL
LIN {X 0,Y 199.87,Z 285.537,A -85,B 0,C 180,E1 -23263.898,E2 -23263.898} C_VEL
LIN {X 0,Y 197.49,Z 297.915,A -85,B 0,C 180,E1 -23264.98,E2 -23264.98} C_VEL
LIN {X 0,Y 194.725,Z 308.825,A -85,B 0,C 180,E1 -23266.281,E2 -23266.281} C_VEL
LIN {X 0,Y 190.979,Z 320.711,A -85,B 0,C 180,E1 -23268.162,E2 -23268.162} C_VEL
LIN {X 0,Y 187.046,Z 331.118,A -85,B 0,C 180,E1 -23270.299,E2 -23270.299} C_VEL
LIN {X 0,Y 182.913,Z 340.44,A -85,B 0,C 180,E1 -23272.758,E2 -23272.758} C_VEL
LIN {X 0,Y 179.008,Z 348.553,A -85,B 0,C 180,E1 -23275.536,E2 -23275.536} C_VEL
LIN {X 0,Y 175.361,Z 355.541,A -85,B 0,C 180,E1 -23278.598,E2 -23278.598} C_VEL
LIN {X 0,Y 171.753,Z 361.515,A -85,B 0,C 180,E1 -23281.927,E2 -23281.927} C_VEL
LIN {X 0,Y 168.791,Z 366.218,A -85,B 0,C 180,E1 -23285.392,E2 -23285.392} C_VEL
LIN {X 0,Y 166.371,Z 369.799,A -85,B 0,C 180,E1 -23288.955,E2 -23288.955} C_VEL
LIN {X 0,Y 164.47,Z 372.361,A -85,B 0,C 180,E1 -23292.593,E2 -23292.593} C_VEL
LIN {X 0,Y 163.512,Z 373.559,A -85,B 0,C 180,E1 -23295.053,E2 -23295.053} C_VEL
LIN {X 0,Y 162.858,Z 374.325,A -85,B 0,C 180,E1 -23297.537,E2 -23297.537} C_VEL
LIN {X 0,Y 162.184,Z 374.657,A -85,B 0,C 180,E1 -23302.528,E2 -23302.528} C_VEL
LIN {X 0,Y 162.13,Z 374.109,A -85,B 0,C 180,E1 -23305.571,E2 -23305.571} C_VEL
LIN {X 0,Y 162.32,Z 372.225,A -85,B 0,C 180,E1 -23309.998,E2 -23309.998} C_VEL
LIN {X 0,Y 162.924,Z 369.644,A -85,B 0,C 180,E1 -23313.708,E2 -23313.708} C_VEL
LIN {X 0,Y 163.955,Z 366.072,A -85,B 0,C 180,E1 -23317.386,E2 -23317.386} C_VEL
LIN {X 0,Y 165.551,Z 361.399,A -85,B 0,C 180,E1 -23321.011,E2 -23321.011} C_VEL
LIN {X 0,Y 168.065,Z 354.38,A -85,B 0,C 180,E1 -23325.148,E2 -23325.148} C_VEL
LIN {X 0,Y 170.912,Z 346.749,A -85,B 0,C 180,E1 -23328.581,E2 -23328.581} C_VEL
LIN {X 0,Y 173.492,Z 338.954,A -85,B 0,C 180,E1 -23331.379,E2 -23331.379} C_VEL
LIN {X 0,Y 176.492,Z 329.436,A -85,B 0,C 180,E1 -23334.087,E2 -23334.087} C_VEL
LIN {X 0,Y 179.484,Z 318.868,A -85,B 0,C 180,E1 -23336.447,E2 -23336.447} C_VEL
LIN {X 0,Y 181.923,Z 308.665,A -85,B 0,C 180,E1 -23338.242,E2 -23338.242} C_VEL
LIN {X 0,Y 184.315,Z 296.526,A -85,B 0,C 180,E1 -23339.87,E2 -23339.87} C_VEL
LIN {X 0,Y 186.181,Z 283.767,A -85,B 0,C 180,E1 -23341.107,E2 -23341.107} C_VEL
LIN {X 0,Y 187.505,Z 270.57,A -85,B 0,C 180,E1 -23341.947,E2 -23341.947} C_VEL
LIN {X 0,Y 190.238,Z 218.184,A -85,B 0,C 180,E1 -23343.808,E2 -23343.808} C_VEL
LIN {X 0,Y 183.639,Z 204.458,A -85,B 0,C 180,E1 -23346.037,E2 -23346.037} C_VEL
LIN {X 0,Y 176.864,Z 192.694,A -85,B 0,C 180,E1 -23348.46,E2 -23348.46} C_VEL
LIN {X 0,Y 172.054,Z 185.274,A -85,B 0,C 180,E1 -23350.304,E2 -23350.304} C_VEL
LIN {X 0,Y 169.432,Z 181.397,A -85,B 0,C 180,E1 -23351.369,E2 -23351.369} C_VEL
LIN {X 0,Y 166.985,Z 177.755,A -85,B 0,C 180,E1 -23352.412,E2 -23352.412} C_VEL
LIN {X 0,Y 164.962,Z 175.314,A -85,B 0,C 180,E1 -23353.278,E2 -23353.278} C_VEL
LIN {X 0,Y 164.26,Z 173.021,A -85,B 0,C 180,E1 -23353.724,E2 -23353.724} C_VEL
LIN {X 0,Y 164.259,Z 173.017,A -85,B 0,C 180,E1 -23356.797,E2 -23356.797} C_VEL
LIN {X 0,Y 164.29,Z 173.02,A -85,B 0,C 180,E1 -23360.35,E2 -23360.35} C_VEL
LIN {X 0,Y 164.324,Z 173.018,A -85,B 0,C 180,E1 -23364.347,E2 -23364.347} C_VEL
LIN {X 0,Y 164.383,Z 173.009,A -85,B 0,C 180,E1 -23369.133,E2 -23369.133} C_VEL
LIN {X 0,Y 164.399,Z 173.006,A -85,B 0,C 180,E1 -23374.691,E2 -23374.691} C_VEL
LIN {X 0,Y 164.431,Z 172.998,A -85,B 0,C 180,E1 -23380.094,E2 -23380.094} C_VEL
LIN {X 0,Y 164.477,Z 172.985,A -85,B 0,C 180,E1 -23385.145,E2 -23385.145} C_VEL
LIN {X 0,Y 164.755,Z 172.945,A -85,B 0,C 180,E1 -23390.175,E2 -23390.175} C_VEL
LIN {X 0,Y 164.809,Z 172.905,A -85,B 0,C 180,E1 -23392.65,E2 -23392.65} C_VEL
LIN {X 0,Y 165.264,Z 172.899,A -85,B 0,C 180,E1 -23400,E2 -23400} C_VEL
LIN {X 0,Y 164.809,Z 172.95,A -85,B 0,C 180,E1 -23407.35,E2 -23407.35} C_VEL
LIN {X 0,Y 164.693,Z 172.967,A -85,B 0,C 180,E1 -23411.058,E2 -23411.058} C_VEL
LIN {X 0,Y 164.443,Z 173.002,A -85,B 0,C 180,E1 -23417.407,E2 -23417.407} C_VEL
LIN {X 0,Y 164.441,Z 173.002,A -85,B 0,C 180,E1 -23419.993,E2 -23419.993} C_VEL
LIN {X 0,Y 164.378,Z 173.014,A -85,B 0,C 180,E1 -23426.129,E2 -23426.129} C_VEL
LIN {X 0,Y 164.367,Z 173.016,A -85,B 0,C 180,E1 -23431.228,E2 -23431.228} C_VEL
LIN {X 0,Y 164.288,Z 173.025,A -85,B 0,C 180,E1 -23436.791,E2 -23436.791} C_VEL
LIN {X 0,Y 164.289,Z 173.143,A -85,B 0,C 180,E1 -23439.65,E2 -23439.65} C_VEL
LIN {X 0,Y 164.979,Z 175.312,A -85,B 0,C 180,E1 -23441.119,E2 -23441.119} C_VEL
LIN {X 0,Y 167.455,Z 179.56,A -85,B 0,C 180,E1 -23442.249,E2 -23442.249} C_VEL
LIN {X 0,Y 169.028,Z 182.188,A -85,B 0,C 180,E1 -23442.934,E2 -23442.934} C_VEL
LIN {X 0,Y 174.133,Z 191.227,A -85,B 0,C 180,E1 -23445.052,E2 -23445.052} C_VEL
LIN {X 0,Y 180.059,Z 203.008,A -85,B 0,C 180,E1 -23447.35,E2 -23447.35} C_VEL
LIN {X 0,Y 185.719,Z 216.749,A -85,B 0,C 180,E1 -23449.463,E2 -23449.463} C_VEL
LIN {X 0,Y 187.404,Z 221.878,A -85,B 0,C 180,E1 -23450.106,E2 -23450.106} C_VEL
LIN {X 0,Y 189.101,Z 241.163,A -85,B 0,C 180,E1 -23451.388,E2 -23451.388} C_VEL
LIN {X 0,Y 186.728,Z 285.384,A -85,B 0,C 180,E1 -23452.975,E2 -23452.975} C_VEL
LIN {X 0,Y 185.261,Z 298.6,A -85,B 0,C 180,E1 -23453.82,E2 -23453.82} C_VEL
LIN {X 0,Y 183.075,Z 311.292,A -85,B 0,C 180,E1 -23455.013,E2 -23455.013} C_VEL
LIN {X 0,Y 180.432,Z 323.365,A -85,B 0,C 180,E1 -23456.624,E2 -23456.624} C_VEL
LIN {X 0,Y 177.902,Z 332.971,A -85,B 0,C 180,E1 -23458.281,E2 -23458.281} C_VEL
LIN {X 0,Y 176,Z 337.875,A -85,B 0,C 180,E1 -23459.208,E2 -23459.208} C_VEL
LIN {X 0,Y 171.042,Z 345.406,A -85,B 0,C 180,E1 -23460.604,E2 -23460.604} C_VEL
LIN {X 0,Y 165.979,Z 352.361,A -85,B 0,C 180,E1 -23462.252,E2 -23462.252} C_VEL
LIN {X 0,Y 163.955,Z 356.372,A -85,B 0,C 180,E1 -23463.549,E2 -23463.549} C_VEL
LIN {X 0,Y 161.193,Z 364.503,A -85,B 0,C 180,E1 -23466.899,E2 -23466.899} C_VEL
LIN {X 0,Y 158.678,Z 371.54,A -85,B 0,C 180,E1 -23470.602,E2 -23470.602} C_VEL
LIN {X 0,Y 156.681,Z 377.168,A -85,B 0,C 180,E1 -23474.39,E2 -23474.39} C_VEL
LIN {X 0,Y 155.525,Z 381.602,A -85,B 0,C 180,E1 -23478.27,E2 -23478.27} C_VEL
LIN {X 0,Y 154.959,Z 384.948,A -85,B 0,C 180,E1 -23482.183,E2 -23482.183} C_VEL
LIN {X 0,Y 154.875,Z 387.55,A -85,B 0,C 180,E1 -23486.684,E2 -23486.684} C_VEL
LIN {X 0,Y 155.059,Z 388.693,A -85,B 0,C 180,E1 -23490.002,E2 -23490.002} C_VEL
LIN {X 0,Y 154.836,Z 389.087,A -85,B 0,C 180,E1 -23493.057,E2 -23493.057} C_VEL
LIN {X 0,Y 154.917,Z 388.646,A -85,B 0,C 180,E1 -23497.824,E2 -23497.824} C_VEL
LIN {X 0,Y 155.309,Z 387.854,A -85,B 0,C 180,E1 -23500.431,E2 -23500.431} C_VEL
LIN {X 0,Y 156.87,Z 384.992,A -85,B 0,C 180,E1 -23505.596,E2 -23505.596} C_VEL
LIN {X 0,Y 158.965,Z 381.747,A -85,B 0,C 180,E1 -23509.367,E2 -23509.367} C_VEL
LIN {X 0,Y 161.689,Z 377.45,A -85,B 0,C 180,E1 -23513.031,E2 -23513.031} C_VEL
LIN {X 0,Y 165.027,Z 371.829,A -85,B 0,C 180,E1 -23516.668,E2 -23516.668} C_VEL
LIN {X 0,Y 168.786,Z 365.171,A -85,B 0,C 180,E1 -23519.98,E2 -23519.98} C_VEL
LIN {X 0,Y 173.417,Z 356.727,A -85,B 0,C 180,E1 -23523.171,E2 -23523.171} C_VEL
LIN {X 0,Y 177.709,Z 348.047,A -85,B 0,C 180,E1 -23525.687,E2 -23525.687} C_VEL
LIN {X 0,Y 182.33,Z 337.38,A -85,B 0,C 180,E1 -23528.08,E2 -23528.08} C_VEL
LIN {X 0,Y 186.355,Z 326.788,A -85,B 0,C 180,E1 -23529.877,E2 -23529.877} C_VEL
LIN {X 0,Y 190.048,Z 314.981,A -85,B 0,C 180,E1 -23531.379,E2 -23531.379} C_VEL
LIN {X 0,Y 193.008,Z 302.717,A -85,B 0,C 180,E1 -23532.527,E2 -23532.527} C_VEL
LIN {X 0,Y 195.2,Z 289.692,A -85,B 0,C 180,E1 -23533.39,E2 -23533.39} C_VEL
LIN {X 0,Y 196.552,Z 275.74,A -85,B 0,C 180,E1 -23533.936,E2 -23533.936} C_VEL
LIN {X 0,Y 198.262,Z 247.996,A -85,B 0,C 180,E1 -23534.85,E2 -23534.85} C_VEL
LIN {X 0,Y 197.665,Z 242.788,A -85,B 0,C 180,E1 -23535.307,E2 -23535.307} C_VEL
LIN {X 0,Y 192.695,Z 230.239,A -85,B 0,C 180,E1 -23537.638,E2 -23537.638} C_VEL
LIN {X 0,Y 188.09,Z 220.322,A -85,B 0,C 180,E1 -23539.918,E2 -23539.918} C_VEL
LIN {X 0,Y 182.904,Z 210.604,A -85,B 0,C 180,E1 -23542.688,E2 -23542.688} C_VEL
LIN {X 0,Y 178.641,Z 203.027,A -85,B 0,C 180,E1 -23545.219,E2 -23545.219} C_VEL
LIN {X 0,Y 174.845,Z 197.006,A -85,B 0,C 180,E1 -23547.686,E2 -23547.686} C_VEL
LIN {X 0,Y 171.231,Z 191.512,A -85,B 0,C 180,E1 -23550.311,E2 -23550.311} C_VEL
LIN {X 0,Y 167.417,Z 186.195,A -85,B 0,C 180,E1 -23553.458,E2 -23553.458} C_VEL
LIN {X 0,Y 166.818,Z 185.355,A -85,B 0,C 180,E1 -23554.001,E2 -23554.001} C_VEL
LIN {X 0,Y 164.12,Z 183.019,A -85,B 0,C 180,E1 -23556.498,E2 -23556.498} C_VEL
LIN {X 0,Y 162.648,Z 180.35,A -85,B 0,C 180,E1 -23558.202,E2 -23558.202} C_VEL
LIN {X 0,Y 162.484,Z 179.846,A -85,B 0,C 180,E1 -23558.429,E2 -23558.429} C_VEL
LIN {X 0,Y 159.481,Z 178.112,A -85,B 0,C 180,E1 -23562.033,E2 -23562.033} C_VEL
LIN {X 0,Y 157.852,Z 175.605,A -85,B 0,C 180,E1 -23564.754,E2 -23564.754} C_VEL
LIN {X 0,Y 157.447,Z 173.853,A -85,B 0,C 180,E1 -23565.871,E2 -23565.871} C_VEL
LIN {X 0,Y 157.688,Z 173.832,A -85,B 0,C 180,E1 -23569.731,E2 -23569.731} C_VEL
LIN {X 0,Y 157.757,Z 173.817,A -85,B 0,C 180,E1 -23572.32,E2 -23572.32} C_VEL
LIN {X 0,Y 158.234,Z 173.776,A -85,B 0,C 180,E1 -23580,E2 -23580} C_VEL
LIN {X 0,Y 157.761,Z 173.817,A -85,B 0,C 180,E1 -23587.681,E2 -23587.681} C_VEL
LIN {X 0,Y 157.722,Z 173.968,A -85,B 0,C 180,E1 -23590.385,E2 -23590.385} C_VEL
LIN {X 0,Y 158.433,Z 176.482,A -85,B 0,C 180,E1 -23591.954,E2 -23591.954} C_VEL
LIN {X 0,Y 160.204,Z 178.646,A -85,B 0,C 180,E1 -23594.611,E2 -23594.611} C_VEL
LIN {X 0,Y 162.659,Z 180.025,A -85,B 0,C 180,E1 -23597.443,E2 -23597.443} C_VEL
LIN {X 0,Y 164.15,Z 183.027,A -85,B 0,C 180,E1 -23599.206,E2 -23599.206} C_VEL
LIN {X 0,Y 166.464,Z 185.128,A -85,B 0,C 180,E1 -23601.373,E2 -23601.373} C_VEL
LIN {X 0,Y 167.237,Z 185.712,A -85,B 0,C 180,E1 -23602.032,E2 -23602.032} C_VEL
LIN {X 0,Y 169.439,Z 189.113,A -85,B 0,C 180,E1 -23603.956,E2 -23603.956} C_VEL
LIN {X 0,Y 171.435,Z 191.075,A -85,B 0,C 180,E1 -23605.456,E2 -23605.456} C_VEL
LIN {X 0,Y 173.928,Z 194.543,A -85,B 0,C 180,E1 -23607.266,E2 -23607.266} C_VEL
LIN {X 0,Y 175.455,Z 196.394,A -85,B 0,C 180,E1 -23608.281,E2 -23608.281} C_VEL
LIN {X 0,Y 179.23,Z 201.638,A -85,B 0,C 180,E1 -23610.648,E2 -23610.648} C_VEL
LIN {X 0,Y 183.755,Z 208.021,A -85,B 0,C 180,E1 -23613.19,E2 -23613.19} C_VEL
LIN {X 0,Y 190.445,Z 218.609,A -85,B 0,C 180,E1 -23616.553,E2 -23616.553} C_VEL
LIN {X 0,Y 196.558,Z 229.636,A -85,B 0,C 180,E1 -23619.312,E2 -23619.312} C_VEL
LIN {X 0,Y 199.134,Z 234.734,A -85,B 0,C 180,E1 -23620.406,E2 -23620.406} C_VEL
LIN {X 0,Y 196.629,Z 272.341,A -85,B 0,C 180,E1 -23621.672,E2 -23621.672} C_VEL
LIN {X 0,Y 194.791,Z 285.877,A -85,B 0,C 180,E1 -23622.468,E2 -23622.468} C_VEL
LIN {X 0,Y 192.244,Z 298.536,A -85,B 0,C 180,E1 -23623.588,E2 -23623.588} C_VEL
LIN {X 0,Y 189.063,Z 310.44,A -85,B 0,C 180,E1 -23625.065,E2 -23625.065} C_VEL
LIN {X 0,Y 185.231,Z 321.846,A -85,B 0,C 180,E1 -23626.923,E2 -23626.923} C_VEL
LIN {X 0,Y 181.162,Z 332.096,A -85,B 0,C 180,E1 -23629.105,E2 -23629.105} C_VEL
LIN {X 0,Y 177.267,Z 340.459,A -85,B 0,C 180,E1 -23631.358,E2 -23631.358} C_VEL
LIN {X 0,Y 172.815,Z 349.211,A -85,B 0,C 180,E1 -23634.426,E2 -23634.426} C_VEL
LIN {X 0,Y 168.605,Z 356.772,A -85,B 0,C 180,E1 -23637.894,E2 -23637.894} C_VEL
LIN {X 0,Y 165.469,Z 361.672,A -85,B 0,C 180,E1 -23640.76,E2 -23640.76} C_VEL
LIN {X 0,Y 162.312,Z 366.41,A -85,B 0,C 180,E1 -23644.34,E2 -23644.34} C_VEL
LIN {X 0,Y 160.295,Z 369.187,A -85,B 0,C 180,E1 -23647.034,E2 -23647.034} C_VEL
LIN {X 0,Y 157.649,Z 372.62,A -85,B 0,C 180,E1 -23651.814,E2 -23651.814} C_VEL
LIN {X 0,Y 156.603,Z 373.832,A -85,B 0,C 180,E1 -23654.377,E2 -23654.377} C_VEL
LIN {X 0,Y 155.873,Z 374.629,A -85,B 0,C 180,E1 -23656.969,E2 -23656.969} C_VEL
LIN {X 0,Y 155.133,Z 374.989,A -85,B 0,C 180,E1 -23662.187,E2 -23662.187} C_VEL
LIN {X 0,Y 155.035,Z 374.338,A -85,B 0,C 180,E1 -23665.794,E2 -23665.794} C_VEL
LIN {X 0,Y 155.234,Z 372.616,A -85,B 0,C 180,E1 -23669.998,E2 -23669.998} C_VEL
LIN {X 0,Y 155.872,Z 370.065,A -85,B 0,C 180,E1 -23673.876,E2 -23673.876} C_VEL
LIN {X 0,Y 156.95,Z 366.527,A -85,B 0,C 180,E1 -23677.718,E2 -23677.718} C_VEL
LIN {X 0,Y 158.621,Z 361.889,A -85,B 0,C 180,E1 -23681.498,E2 -23681.498} C_VEL
LIN {X 0,Y 161.248,Z 354.91,A -85,B 0,C 180,E1 -23685.805,E2 -23685.805} C_VEL
LIN {X 0,Y 164.097,Z 347.734,A -85,B 0,C 180,E1 -23689.195,E2 -23689.195} C_VEL
LIN {X 0,Y 166.936,Z 339.605,A -85,B 0,C 180,E1 -23692.263,E2 -23692.263} C_VEL
LIN {X 0,Y 170.408,Z 329.093,A -85,B 0,C 180,E1 -23695.331,E2 -23695.331} C_VEL
LIN {X 0,Y 173.535,Z 318.389,A -85,B 0,C 180,E1 -23697.755,E2 -23697.755} C_VEL
LIN {X 0,Y 176.137,Z 307.968,A -85,B 0,C 180,E1 -23699.586,E2 -23699.586} C_VEL
LIN {X 0,Y 178.634,Z 295.443,A -85,B 0,C 180,E1 -23701.251,E2 -23701.251} C_VEL
LIN {X 0,Y 180.496,Z 282.948,A -85,B 0,C 180,E1 -23702.45,E2 -23702.45} C_VEL
LIN {X 0,Y 181.776,Z 270.072,A -85,B 0,C 180,E1 -23703.253,E2 -23703.253} C_VEL
LIN {X 0,Y 184.489,Z 220.281,A -85,B 0,C 180,E1 -23705.053,E2 -23705.053} C_VEL
LIN {X 0,Y 177.907,Z 206.724,A -85,B 0,C 180,E1 -23707.431,E2 -23707.431} C_VEL
LIN {X 0,Y 170.523,Z 194.043,A -85,B 0,C 180,E1 -23710.291,E2 -23710.291} C_VEL
LIN {X 0,Y 164.924,Z 185.725,A -85,B 0,C 180,E1 -23712.653,E2 -23712.653} C_VEL
LIN {X 0,Y 163.186,Z 183.147,A -85,B 0,C 180,E1 -23713.44,E2 -23713.44} C_VEL
LIN {X 0,Y 160.831,Z 179.834,A -85,B 0,C 180,E1 -23714.542,E2 -23714.542} C_VEL
LIN {X 0,Y 160.182,Z 178.825,A -85,B 0,C 180,E1 -23714.861,E2 -23714.861} C_VEL
LIN {X 0,Y 158.159,Z 176.637,A -85,B 0,C 180,E1 -23715.823,E2 -23715.823} C_VEL
LIN {X 0,Y 157.238,Z 173.893,A -85,B 0,C 180,E1 -23716.45,E2 -23716.45} C_VEL
LIN {X 0,Y 157.201,Z 173.897,A -85,B 0,C 180,E1 -23721.251,E2 -23721.251} C_VEL
LIN {X 0,Y 157.273,Z 173.896,A -85,B 0,C 180,E1 -23724.484,E2 -23724.484} C_VEL
LIN {X 0,Y 157.286,Z 173.886,A -85,B 0,C 180,E1 -23728.094,E2 -23728.094} C_VEL
LIN {X 0,Y 157.307,Z 173.881,A -85,B 0,C 180,E1 -23733.463,E2 -23733.463} C_VEL
LIN {X 0,Y 157.37,Z 173.874,A -85,B 0,C 180,E1 -23739.683,E2 -23739.683} C_VEL
LIN {X 0,Y 157.413,Z 173.863,A -85,B 0,C 180,E1 -23744.461,E2 -23744.461} C_VEL
LIN {X 0,Y 157.678,Z 173.831,A -85,B 0,C 180,E1 -23749.73,E2 -23749.73} C_VEL
LIN {X 0,Y 157.748,Z 173.785,A -85,B 0,C 180,E1 -23752.319,E2 -23752.319} C_VEL
LIN {X 0,Y 158.226,Z 173.775,A -85,B 0,C 180,E1 -23760,E2 -23760} C_VEL
LIN {X 0,Y 157.748,Z 173.83,A -85,B 0,C 180,E1 -23767.681,E2 -23767.681} C_VEL
LIN {X 0,Y 157.623,Z 173.847,A -85,B 0,C 180,E1 -23771.227,E2 -23771.227} C_VEL
LIN {X 0,Y 157.412,Z 173.877,A -85,B 0,C 180,E1 -23775.538,E2 -23775.538} C_VEL
LIN {X 0,Y 157.349,Z 173.884,A -85,B 0,C 180,E1 -23780.936,E2 -23780.936} C_VEL
LIN {X 0,Y 157.302,Z 173.898,A -85,B 0,C 180,E1 -23786.682,E2 -23786.682} C_VEL
LIN {X 0,Y 157.268,Z 173.902,A -85,B 0,C 180,E1 -23792.429,E2 -23792.429} C_VEL
LIN {X 0,Y 157.309,Z 174.072,A -85,B 0,C 180,E1 -23797.768,E2 -23797.768} C_VEL
LIN {X 0,Y 157.426,Z 174.663,A -85,B 0,C 180,E1 -23798.128,E2 -23798.128} C_VEL
LIN {X 0,Y 158.586,Z 177.225,A -85,B 0,C 180,E1 -23798.783,E2 -23798.783} C_VEL
LIN {X 0,Y 161.414,Z 181.083,A -85,B 0,C 180,E1 -23800.155,E2 -23800.155} C_VEL
LIN {X 0,Y 165.098,Z 187.334,A -85,B 0,C 180,E1 -23801.897,E2 -23801.897} C_VEL
LIN {X 0,Y 169.933,Z 196.105,A -85,B 0,C 180,E1 -23804.029,E2 -23804.029} C_VEL
LIN {X 0,Y 175.923,Z 208.408,A -85,B 0,C 180,E1 -23806.496,E2 -23806.496} C_VEL
LIN {X 0,Y 181.627,Z 222.966,A -85,B 0,C 180,E1 -23808.76,E2 -23808.76} C_VEL
LIN {X 0,Y 183.108,Z 237.607,A -85,B 0,C 180,E1 -23809.843,E2 -23809.843} C_VEL
LIN {X 0,Y 183.311,Z 243.249,A -85,B 0,C 180,E1 -23810.164,E2 -23810.164} C_VEL
LIN {X 0,Y 180.967,Z 284.711,A -85,B 0,C 180,E1 -23811.676,E2 -23811.676} C_VEL
LIN {X 0,Y 179.416,Z 298.038,A -85,B 0,C 180,E1 -23812.531,E2 -23812.531} C_VEL
LIN {X 0,Y 177.492,Z 309.091,A -85,B 0,C 180,E1 -23813.566,E2 -23813.566} C_VEL
LIN {X 0,Y 174.92,Z 320.835,A -85,B 0,C 180,E1 -23815.075,E2 -23815.075} C_VEL
LIN {X 0,Y 172.061,Z 331.529,A -85,B 0,C 180,E1 -23816.889,E2 -23816.889} C_VEL
LIN {X 0,Y 168.711,Z 342.456,A -85,B 0,C 180,E1 -23819.319,E2 -23819.319} C_VEL
LIN {X 0,Y 165.362,Z 352.268,A -85,B 0,C 180,E1 -23822.13,E2 -23822.13} C_VEL
LIN {X 0,Y 163.955,Z 356.372,A -85,B 0,C 180,E1 -23823.549,E2 -23823.549} C_VEL
LIN {X 0,Y 162.01,Z 360.257,A -85,B 0,C 180,E1 -23824.957,E2 -23824.957} C_VEL
LIN {X 0,Y 157.214,Z 366.075,A -85,B 0,C 180,E1 -23827.271,E2 -23827.271} C_VEL
LIN {X 0,Y 152.516,Z 371.245,A -85,B 0,C 180,E1 -23829.887,E2 -23829.887} C_VEL
LIN {X 0,Y 150.782,Z 374.113,A -85,B 0,C 180,E1 -23831.733,E2 -23831.733} C_VEL
LIN {X 0,Y 148.904,Z 379.809,A -85,B 0,C 180,E1 -23836.353,E2 -23836.353} C_VEL
LIN {X 0,Y 148.075,Z 383.535,A -85,B 0,C 180,E1 -23840.44,E2 -23840.44} C_VEL
LIN {X 0,Y 147.747,Z 386.226,A -85,B 0,C 180,E1 -23844.543,E2 -23844.543} C_VEL
LIN {X 0,Y 147.803,Z 387.493,A -85,B 0,C 180,E1 -23847.277,E2 -23847.277} C_VEL
LIN {X 0,Y 147.963,Z 388.347,A -85,B 0,C 180,E1 -23850.002,E2 -23850.002} C_VEL
LIN {X 0,Y 147.773,Z 388.742,A -85,B 0,C 180,E1 -23852.866,E2 -23852.866} C_VEL
LIN {X 0,Y 147.866,Z 388.341,A -85,B 0,C 180,E1 -23858.2,E2 -23858.2} C_VEL
LIN {X 0,Y 148.302,Z 387.567,A -85,B 0,C 180,E1 -23860.929,E2 -23860.929} C_VEL
LIN {X 0,Y 149.015,Z 386.358,A -85,B 0,C 180,E1 -23863.642,E2 -23863.642} C_VEL
LIN {X 0,Y 150.675,Z 383.797,A -85,B 0,C 180,E1 -23867.651,E2 -23867.651} C_VEL
LIN {X 0,Y 153.13,Z 380.245,A -85,B 0,C 180,E1 -23871.543,E2 -23871.543} C_VEL
LIN {X 0,Y 156.264,Z 375.607,A -85,B 0,C 180,E1 -23875.296,E2 -23875.296} C_VEL
LIN {X 0,Y 159.851,Z 369.738,A -85,B 0,C 180,E1 -23878.925,E2 -23878.925} C_VEL
LIN {X 0,Y 164.213,Z 362.439,A -85,B 0,C 180,E1 -23882.344,E2 -23882.344} C_VEL
LIN {X 0,Y 169.267,Z 353.406,A -85,B 0,C 180,E1 -23885.543,E2 -23885.543} C_VEL
LIN {X 0,Y 173.909,Z 344.095,A -85,B 0,C 180,E1 -23888.047,E2 -23888.047} C_VEL
LIN {X 0,Y 178.355,Z 333.751,A -85,B 0,C 180,E1 -23890.186,E2 -23890.186} C_VEL
LIN {X 0,Y 182.614,Z 322.286,A -85,B 0,C 180,E1 -23891.968,E2 -23891.968} C_VEL
LIN {X 0,Y 186.147,Z 310.293,A -85,B 0,C 180,E1 -23893.369,E2 -23893.369} C_VEL
LIN {X 0,Y 188.948,Z 297.719,A -85,B 0,C 180,E1 -23894.408,E2 -23894.408} C_VEL
LIN {X 0,Y 190.958,Z 284.195,A -85,B 0,C 180,E1 -23895.159,E2 -23895.159} C_VEL
LIN {X 0,Y 193.418,Z 249.16,A -85,B 0,C 180,E1 -23896.34,E2 -23896.34} C_VEL
LIN {X 0,Y 192.989,Z 245.732,A -85,B 0,C 180,E1 -23896.672,E2 -23896.672} C_VEL
LIN {X 0,Y 188.427,Z 233.871,A -85,B 0,C 180,E1 -23898.976,E2 -23898.976} C_VEL
LIN {X 0,Y 182.989,Z 222.084,A -85,B 0,C 180,E1 -23901.893,E2 -23901.893} C_VEL
LIN {X 0,Y 177.679,Z 212.092,A -85,B 0,C 180,E1 -23905.038,E2 -23905.038} C_VEL
LIN {X 0,Y 172.685,Z 203.454,A -85,B 0,C 180,E1 -23908.4,E2 -23908.4} C_VEL
LIN {X 0,Y 168.758,Z 197.41,A -85,B 0,C 180,E1 -23911.406,E2 -23911.406} C_VEL
LIN {X 0,Y 164.951,Z 191.946,A -85,B 0,C 180,E1 -23914.782,E2 -23914.782} C_VEL
LIN {X 0,Y 162.23,Z 189.315,A -85,B 0,C 180,E1 -23917.473,E2 -23917.473} C_VEL
LIN {X 0,Y 160.724,Z 186.603,A -85,B 0,C 180,E1 -23919.336,E2 -23919.336} C_VEL
LIN {X 0,Y 157.907,Z 184.582,A -85,B 0,C 180,E1 -23923.018,E2 -23923.018} C_VEL
LIN {X 0,Y 156.458,Z 182.073,A -85,B 0,C 180,E1 -23925.697,E2 -23925.697} C_VEL
LIN {X 0,Y 156.077,Z 180.79,A -85,B 0,C 180,E1 -23926.658,E2 -23926.658} C_VEL
LIN {X 0,Y 153.327,Z 179.111,A -85,B 0,C 180,E1 -23938.687,E2 -23938.687} C_VEL
LIN {X 0,Y 153.573,Z 179.287,A -85,B 0,C 180,E1 -23941.311,E2 -23941.311} C_VEL
LIN {X 0,Y 156.385,Z 180.998,A -85,B 0,C 180,E1 -23949.621,E2 -23949.621} C_VEL
LIN {X 0,Y 157.381,Z 183.712,A -85,B 0,C 180,E1 -23951.756,E2 -23951.756} C_VEL
LIN {X 0,Y 159.588,Z 185.991,A -85,B 0,C 180,E1 -23954.995,E2 -23954.995} C_VEL
LIN {X 0,Y 161.048,Z 186.923,A -85,B 0,C 180,E1 -23956.723,E2 -23956.723} C_VEL
LIN {X 0,Y 162.844,Z 190.081,A -85,B 0,C 180,E1 -23958.868,E2 -23958.868} C_VEL
LIN {X 0,Y 165.416,Z 192.469,A -85,B 0,C 180,E1 -23961.323,E2 -23961.323} C_VEL
LIN {X 0,Y 167.901,Z 196.018,A -85,B 0,C 180,E1 -23963.542,E2 -23963.542} C_VEL
LIN {X 0,Y 169.406,Z 197.703,A -85,B 0,C 180,E1 -23964.732,E2 -23964.732} C_VEL
LIN {X 0,Y 173.121,Z 202.725,A -85,B 0,C 180,E1 -23967.469,E2 -23967.469} C_VEL
LIN {X 0,Y 176.388,Z 207.312,A -85,B 0,C 180,E1 -23969.625,E2 -23969.625} C_VEL
LIN {X 0,Y 180.873,Z 213.912,A -85,B 0,C 180,E1 -23972.295,E2 -23972.295} C_VEL
LIN {X 0,Y 186.535,Z 223.141,A -85,B 0,C 180,E1 -23975.318,E2 -23975.318} C_VEL
LIN {X 0,Y 191.825,Z 232.755,A -85,B 0,C 180,E1 -23977.873,E2 -23977.873} C_VEL
LIN {X 0,Y 194.181,Z 237.344,A -85,B 0,C 180,E1 -23978.942,E2 -23978.942} C_VEL
LIN {X 0,Y 191.77,Z 272.442,A -85,B 0,C 180,E1 -23980.145,E2 -23980.145} C_VEL
LIN {X 0,Y 189.942,Z 285.672,A -85,B 0,C 180,E1 -23980.925,E2 -23980.925} C_VEL
LIN {X 0,Y 187.396,Z 298.048,A -85,B 0,C 180,E1 -23982.008,E2 -23982.008} C_VEL
LIN {X 0,Y 184.037,Z 310.172,A -85,B 0,C 180,E1 -23983.481,E2 -23983.481} C_VEL
LIN {X 0,Y 180.07,Z 321.688,A -85,B 0,C 180,E1 -23985.368,E2 -23985.368} C_VEL
LIN {X 0,Y 175.808,Z 332.037,A -85,B 0,C 180,E1 -23987.576,E2 -23987.576} C_VEL
LIN {X 0,Y 171.733,Z 340.47,A -85,B 0,C 180,E1 -23989.866,E2 -23989.866} C_VEL
LIN {X 0,Y 167.506,Z 348.494,A -85,B 0,C 180,E1 -23992.677,E2 -23992.677} C_VEL
LIN {X 0,Y 163.307,Z 355.774,A -85,B 0,C 180,E1 -23995.979,E2 -23995.979} C_VEL
LIN {X 0,Y 159.247,Z 361.828,A -85,B 0,C 180,E1 -23999.499,E2 -23999.499} C_VEL
LIN {X 0,Y 155.865,Z 366.604,A -85,B 0,C 180,E1 -24003.196,E2 -24003.196} C_VEL
LIN {X 0,Y 153.493,Z 369.678,A -85,B 0,C 180,E1 -24006.313,E2 -24006.313} C_VEL
LIN {X 0,Y 150.867,Z 372.878,A -85,B 0,C 180,E1 -24010.966,E2 -24010.966} C_VEL
LIN {X 0,Y 149.717,Z 374.106,A -85,B 0,C 180,E1 -24013.639,E2 -24013.639} C_VEL
LIN {X 0,Y 148.915,Z 374.929,A -85,B 0,C 180,E1 -24016.349,E2 -24016.349} C_VEL
LIN {X 0,Y 148.058,Z 375.322,A -85,B 0,C 180,E1 -24021.811,E2 -24021.811} C_VEL
LIN {X 0,Y 147.941,Z 374.565,A -85,B 0,C 180,E1 -24026.048,E2 -24026.048} C_VEL
LIN {X 0,Y 148.149,Z 373.006,A -85,B 0,C 180,E1 -24029.998,E2 -24029.998} C_VEL
LIN {X 0,Y 148.537,Z 371.421,A -85,B 0,C 180,E1 -24032.709,E2 -24032.709} C_VEL
LIN {X 0,Y 149.523,Z 368.247,A -85,B 0,C 180,E1 -24036.746,E2 -24036.746} C_VEL
LIN {X 0,Y 151.048,Z 364.024,A -85,B 0,C 180,E1 -24040.723,E2 -24040.723} C_VEL
LIN {X 0,Y 153.628,Z 357.626,A -85,B 0,C 180,E1 -24045.248,E2 -24045.248} C_VEL
LIN {X 0,Y 156.441,Z 350.784,A -85,B 0,C 180,E1 -24048.917,E2 -24048.917} C_VEL
LIN {X 0,Y 159.826,Z 341.868,A -85,B 0,C 180,E1 -24052.625,E2 -24052.625} C_VEL
LIN {X 0,Y 163.37,Z 331.925,A -85,B 0,C 180,E1 -24055.818,E2 -24055.818} C_VEL
LIN {X 0,Y 166.553,Z 321.759,A -85,B 0,C 180,E1 -24058.338,E2 -24058.338} C_VEL
LIN {X 0,Y 169.609,Z 310.486,A -85,B 0,C 180,E1 -24060.501,E2 -24060.501} C_VEL
LIN {X 0,Y 172.236,Z 298.784,A -85,B 0,C 180,E1 -24062.206,E2 -24062.206} C_VEL
LIN {X 0,Y 174.391,Z 285.913,A -85,B 0,C 180,E1 -24063.561,E2 -24063.561} C_VEL
LIN {X 0,Y 175.958,Z 272.087,A -85,B 0,C 180,E1 -24064.517,E2 -24064.517} C_VEL
LIN {X 0,Y 178.866,Z 222.591,A -85,B 0,C 180,E1 -24066.358,E2 -24066.358} C_VEL
LIN {X 0,Y 172.622,Z 209.774,A -85,B 0,C 180,E1 -24068.774,E2 -24068.774} C_VEL
LIN {X 0,Y 165.737,Z 197.858,A -85,B 0,C 180,E1 -24071.639,E2 -24071.639} C_VEL
LIN {X 0,Y 159.733,Z 188.753,A -85,B 0,C 180,E1 -24074.39,E2 -24074.39} C_VEL
LIN {X 0,Y 157.074,Z 184.908,A -85,B 0,C 180,E1 -24075.712,E2 -24075.712} C_VEL
LIN {X 0,Y 154.453,Z 181.637,A -85,B 0,C 180,E1 -24077.06,E2 -24077.06} C_VEL
LIN {X 0,Y 153.435,Z 179.921,A -85,B 0,C 180,E1 -24077.639,E2 -24077.639} C_VEL
LIN {X 0,Y 151.205,Z 177.74,A -85,B 0,C 180,E1 -24078.841,E2 -24078.841} C_VEL
LIN {X 0,Y 150.217,Z 175.138,A -85,B 0,C 180,E1 -24079.522,E2 -24079.522} C_VEL
LIN {X 0,Y 150.141,Z 174.785,A -85,B 0,C 180,E1 -24079.717,E2 -24079.717} C_VEL
LIN {X 0,Y 150.174,Z 174.771,A -85,B 0,C 180,E1 -24082.705,E2 -24082.705} C_VEL
LIN {X 0,Y 150.208,Z 174.765,A -85,B 0,C 180,E1 -24087.366,E2 -24087.366} C_VEL
LIN {X 0,Y 150.235,Z 174.759,A -85,B 0,C 180,E1 -24092.719,E2 -24092.719} C_VEL
LIN {X 0,Y 150.332,Z 174.747,A -85,B 0,C 180,E1 -24099.219,E2 -24099.219} C_VEL
LIN {X 0,Y 150.32,Z 174.748,A -85,B 0,C 180,E1 -24103.708,E2 -24103.708} C_VEL
LIN {X 0,Y 150.599,Z 174.718,A -85,B 0,C 180,E1 -24109.241,E2 -24109.241} C_VEL
LIN {X 0,Y 150.671,Z 174.668,A -85,B 0,C 180,E1 -24111.956,E2 -24111.956} C_VEL
LIN {X 0,Y 151.187,Z 174.652,A -85,B 0,C 180,E1 -24120,E2 -24120} C_VEL
LIN {X 0,Y 150.671,Z 174.712,A -85,B 0,C 180,E1 -24128.044,E2 -24128.044} C_VEL
LIN {X 0,Y 150.565,Z 174.725,A -85,B 0,C 180,E1 -24131.43,E2 -24131.43} C_VEL
LIN {X 0,Y 150.32,Z 174.758,A -85,B 0,C 180,E1 -24136.291,E2 -24136.291} C_VEL
LIN {X 0,Y 150.331,Z 174.758,A -85,B 0,C 180,E1 -24140.781,E2 -24140.781} C_VEL
LIN {X 0,Y 150.234,Z 174.777,A -85,B 0,C 180,E1 -24147.281,E2 -24147.281} C_VEL
LIN {X 0,Y 150.208,Z 174.781,A -85,B 0,C 180,E1 -24152.633,E2 -24152.633} C_VEL
LIN {X 0,Y 150.23,Z 174.973,A -85,B 0,C 180,E1 -24154.863,E2 -24154.863} C_VEL
LIN {X 0,Y 151.072,Z 177.331,A -85,B 0,C 180,E1 -24155.454,E2 -24155.454} C_VEL
LIN {X 0,Y 152.95,Z 179.542,A -85,B 0,C 180,E1 -24156.503,E2 -24156.503} C_VEL
LIN {X 0,Y 153.921,Z 180.492,A -85,B 0,C 180,E1 -24157.012,E2 -24157.012} C_VEL
LIN {X 0,Y 156.666,Z 184.681,A -85,B 0,C 180,E1 -24158.494,E2 -24158.494} C_VEL
LIN {X 0,Y 161.002,Z 191.998,A -85,B 0,C 180,E1 -24160.695,E2 -24160.695} C_VEL
LIN {X 0,Y 165.96,Z 201.316,A -85,B 0,C 180,E1 -24163.032,E2 -24163.032} C_VEL
LIN {X 0,Y 171.477,Z 213.014,A -85,B 0,C 180,E1 -24165.453,E2 -24165.453} C_VEL
LIN {X 0,Y 176.402,Z 225.881,A -85,B 0,C 180,E1 -24167.544,E2 -24167.544} C_VEL
LIN {X 0,Y 177.727,Z 242.858,A -85,B 0,C 180,E1 -24168.765,E2 -24168.765} C_VEL
LIN {X 0,Y 175.311,Z 284.024,A -85,B 0,C 180,E1 -24170.292,E2 -24170.292} C_VEL
LIN {X 0,Y 173.683,Z 297.478,A -85,B 0,C 180,E1 -24171.16,E2 -24171.16} C_VEL
LIN {X 0,Y 171.844,Z 308.034,A -85,B 0,C 180,E1 -24172.163,E2 -24172.163} C_VEL
LIN {X 0,Y 169.121,Z 319.933,A -85,B 0,C 180,E1 -24173.692,E2 -24173.692} C_VEL
LIN {X 0,Y 166.13,Z 330.749,A -85,B 0,C 180,E1 -24175.544,E2 -24175.544} C_VEL
LIN {X 0,Y 162.653,Z 341.786,A -85,B 0,C 180,E1 -24178.045,E2 -24178.045} C_VEL
LIN {X 0,Y 159.073,Z 351.65,A -85,B 0,C 180,E1 -24180.926,E2 -24180.926} C_VEL
LIN {X 0,Y 155.742,Z 360.779,A -85,B 0,C 180,E1 -24184.395,E2 -24184.395} C_VEL
LIN {X 0,Y 153.206,Z 367.705,A -85,B 0,C 180,E1 -24187.765,E2 -24187.765} C_VEL
LIN {X 0,Y 150.782,Z 374.113,A -85,B 0,C 180,E1 -24191.733,E2 -24191.733} C_VEL
LIN {X 0,Y 149.183,Z 376.772,A -85,B 0,C 180,E1 -24193.664,E2 -24193.664} C_VEL
LIN {X 0,Y 143.573,Z 381.75,A -85,B 0,C 180,E1 -24198.246,E2 -24198.246} C_VEL
LIN {X 0,Y 141.17,Z 384.004,A -85,B 0,C 180,E1 -24201.153,E2 -24201.153} C_VEL
LIN {X 0,Y 140.725,Z 384.92,A -85,B 0,C 180,E1 -24202.698,E2 -24202.698} C_VEL
LIN {X 0,Y 140.721,Z 387.169,A -85,B 0,C 180,E1 -24207.254,E2 -24207.254} C_VEL
LIN {X 0,Y 140.868,Z 387.997,A -85,B 0,C 180,E1 -24210.003,E2 -24210.003} C_VEL
LIN {X 0,Y 140.696,Z 388.405,A -85,B 0,C 180,E1 -24212.866,E2 -24212.866} C_VEL
LIN {X 0,Y 140.817,Z 388.035,A -85,B 0,C 180,E1 -24218.614,E2 -24218.614} C_VEL
LIN {X 0,Y 141.319,Z 387.278,A -85,B 0,C 180,E1 -24221.477,E2 -24221.477} C_VEL
LIN {X 0,Y 142.101,Z 386.092,A -85,B 0,C 180,E1 -24224.32,E2 -24224.32} C_VEL
LIN {X 0,Y 143.899,Z 383.558,A -85,B 0,C 180,E1 -24228.512,E2 -24228.512} C_VEL
LIN {X 0,Y 146.51,Z 380.03,A -85,B 0,C 180,E1 -24232.569,E2 -24232.569} C_VEL
LIN {X 0,Y 149.835,Z 375.424,A -85,B 0,C 180,E1 -24236.464,E2 -24236.464} C_VEL
LIN {X 0,Y 154.346,Z 368.472,A -85,B 0,C 180,E1 -24240.817,E2 -24240.817} C_VEL
LIN {X 0,Y 159.107,Z 360.977,A -85,B 0,C 180,E1 -24244.279,E2 -24244.279} C_VEL
LIN {X 0,Y 163.54,Z 353.349,A -85,B 0,C 180,E1 -24246.99,E2 -24246.99} C_VEL
LIN {X 0,Y 168.381,Z 344.116,A -85,B 0,C 180,E1 -24249.535,E2 -24249.535} C_VEL
LIN {X 0,Y 173.003,Z 333.853,A -85,B 0,C 180,E1 -24251.701,E2 -24251.701} C_VEL
LIN {X 0,Y 177.41,Z 322.483,A -85,B 0,C 180,E1 -24253.498,E2 -24253.498} C_VEL
LIN {X 0,Y 181.069,Z 310.671,A -85,B 0,C 180,E1 -24254.907,E2 -24254.907} C_VEL
LIN {X 0,Y 183.953,Z 298.4,A -85,B 0,C 180,E1 -24255.953,E2 -24255.953} C_VEL
LIN {X 0,Y 186.134,Z 284.607,A -85,B 0,C 180,E1 -24256.739,E2 -24256.739} C_VEL
LIN {X 0,Y 188.709,Z 250.364,A -85,B 0,C 180,E1 -24257.905,E2 -24257.905} C_VEL
LIN {X 0,Y 188.256,Z 248.056,A -85,B 0,C 180,E1 -24258.204,E2 -24258.204} C_VEL
LIN {X 0,Y 183.651,Z 236.112,A -85,B 0,C 180,E1 -24260.712,E2 -24260.712} C_VEL
LIN {X 0,Y 178.979,Z 225.959,A -85,B 0,C 180,E1 -24263.425,E2 -24263.425} C_VEL
LIN {X 0,Y 174.546,Z 217.316,A -85,B 0,C 180,E1 -24266.259,E2 -24266.259} C_VEL
LIN {X 0,Y 170.283,Z 209.547,A -85,B 0,C 180,E1 -24269.329,E2 -24269.329} C_VEL
LIN {X 0,Y 166.568,Z 203.589,A -85,B 0,C 180,E1 -24272.347,E2 -24272.347} C_VEL
LIN {X 0,Y 163.04,Z 198.432,A -85,B 0,C 180,E1 -24275.657,E2 -24275.657} C_VEL
LIN {X 0,Y 160.274,Z 195.413,A -85,B 0,C 180,E1 -24278.613,E2 -24278.613} C_VEL
LIN {X 0,Y 159.217,Z 193.405,A -85,B 0,C 180,E1 -24280.017,E2 -24280.017} C_VEL
LIN {X 0,Y 156.614,Z 191.338,A -85,B 0,C 180,E1 -24283.628,E2 -24283.628} C_VEL
LIN {X 0,Y 155.153,Z 188.695,A -85,B 0,C 180,E1 -24286.535,E2 -24286.535} C_VEL
LIN {X 0,Y 154.912,Z 187.806,A -85,B 0,C 180,E1 -24287.204,E2 -24287.204} C_VEL
LIN {X 0,Y 152.436,Z 186.271,A -85,B 0,C 180,E1 -24297.358,E2 -24297.358} C_VEL
LIN {X 0,Y 152.622,Z 186.227,A -85,B 0,C 180,E1 -24300.66,E2 -24300.66} C_VEL
LIN {X 0,Y 155.147,Z 187.961,A -85,B 0,C 180,E1 -24308.959,E2 -24308.959} C_VEL
LIN {X 0,Y 156.315,Z 190.817,A -85,B 0,C 180,E1 -24311.509,E2 -24311.509} C_VEL
LIN {X 0,Y 158.74,Z 193.136,A -85,B 0,C 180,E1 -24315.077,E2 -24315.077} C_VEL
LIN {X 0,Y 159.477,Z 193.701,A -85,B 0,C 180,E1 -24315.988,E2 -24315.988} C_VEL
LIN {X 0,Y 161.435,Z 196.955,A -85,B 0,C 180,E1 -24318.399,E2 -24318.399} C_VEL
LIN {X 0,Y 163.624,Z 199.123,A -85,B 0,C 180,E1 -24320.59,E2 -24320.59} C_VEL
LIN {X 0,Y 166.369,Z 202.902,A -85,B 0,C 180,E1 -24323.117,E2 -24323.117} C_VEL
LIN {X 0,Y 167.783,Z 204.845,A -85,B 0,C 180,E1 -24324.3,E2 -24324.3} C_VEL
LIN {X 0,Y 170.606,Z 208.653,A -85,B 0,C 180,E1 -24326.468,E2 -24326.468} C_VEL
LIN {X 0,Y 174.78,Z 214.764,A -85,B 0,C 180,E1 -24329.345,E2 -24329.345} C_VEL
LIN {X 0,Y 180.323,Z 223.444,A -85,B 0,C 180,E1 -24332.695,E2 -24332.695} C_VEL
LIN {X 0,Y 186.557,Z 234.6,A -85,B 0,C 180,E1 -24336.029,E2 -24336.029} C_VEL
LIN {X 0,Y 189.446,Z 240.598,A -85,B 0,C 180,E1 -24337.471,E2 -24337.471} C_VEL
LIN {X 0,Y 186.963,Z 273.368,A -85,B 0,C 180,E1 -24338.582,E2 -24338.582} C_VEL
LIN {X 0,Y 184.932,Z 287.129,A -85,B 0,C 180,E1 -24339.419,E2 -24339.419} C_VEL
LIN {X 0,Y 182.126,Z 299.708,A -85,B 0,C 180,E1 -24340.559,E2 -24340.559} C_VEL
LIN {X 0,Y 178.586,Z 311.75,A -85,B 0,C 180,E1 -24342.094,E2 -24342.094} C_VEL
LIN {X 0,Y 174.542,Z 322.83,A -85,B 0,C 180,E1 -24343.965,E2 -24343.965} C_VEL
LIN {X 0,Y 170.11,Z 333.001,A -85,B 0,C 180,E1 -24346.208,E2 -24346.208} C_VEL
LIN {X 0,Y 165.433,Z 342.133,A -85,B 0,C 180,E1 -24348.814,E2 -24348.814} C_VEL
LIN {X 0,Y 160.374,Z 351.006,A -85,B 0,C 180,E1 -24352.153,E2 -24352.153} C_VEL
LIN {X 0,Y 155.919,Z 358.104,A -85,B 0,C 180,E1 -24355.704,E2 -24355.704} C_VEL
LIN {X 0,Y 151.85,Z 363.738,A -85,B 0,C 180,E1 -24359.393,E2 -24359.393} C_VEL
LIN {X 0,Y 148.436,Z 368.156,A -85,B 0,C 180,E1 -24363.267,E2 -24363.267} C_VEL
LIN {X 0,Y 145.618,Z 371.49,A -85,B 0,C 180,E1 -24367.285,E2 -24367.285} C_VEL
LIN {X 0,Y 144.125,Z 373.136,A -85,B 0,C 180,E1 -24370.039,E2 -24370.039} C_VEL
LIN {X 0,Y 141.985,Z 375.224,A -85,B 0,C 180,E1 -24375.668,E2 -24375.668} C_VEL
LIN {X 0,Y 141.005,Z 375.655,A -85,B 0,C 180,E1 -24381.398,E2 -24381.398} C_VEL
LIN {X 0,Y 140.871,Z 374.825,A -85,B 0,C 180,E1 -24386.203,E2 -24386.203} C_VEL
LIN {X 0,Y 141.046,Z 373.398,A -85,B 0,C 180,E1 -24389.997,E2 -24389.997} C_VEL
LIN {X 0,Y 141.46,Z 371.827,A -85,B 0,C 180,E1 -24392.845,E2 -24392.845} C_VEL
LIN {X 0,Y 142.51,Z 368.684,A -85,B 0,C 180,E1 -24397.079,E2 -24397.079} C_VEL
LIN {X 0,Y 144.117,Z 364.496,A -85,B 0,C 180,E1 -24401.246,E2 -24401.246} C_VEL
LIN {X 0,Y 146.83,Z 358.134,A -85,B 0,C 180,E1 -24405.972,E2 -24405.972} C_VEL
LIN {X 0,Y 149.736,Z 351.435,A -85,B 0,C 180,E1 -24409.753,E2 -24409.753} C_VEL
LIN {X 0,Y 153.182,Z 342.856,A -85,B 0,C 180,E1 -24413.504,E2 -24413.504} C_VEL
LIN {X 0,Y 156.71,Z 333.585,A -85,B 0,C 180,E1 -24416.643,E2 -24416.643} C_VEL
LIN {X 0,Y 160.026,Z 323.793,A -85,B 0,C 180,E1 -24419.245,E2 -24419.245} C_VEL
LIN {X 0,Y 163.169,Z 312.962,A -85,B 0,C 180,E1 -24421.48,E2 -24421.48} C_VEL
LIN {X 0,Y 166.066,Z 300.832,A -85,B 0,C 180,E1 -24423.375,E2 -24423.375} C_VEL
LIN {X 0,Y 168.453,Z 288.086,A -85,B 0,C 180,E1 -24424.82,E2 -24424.82} C_VEL
LIN {X 0,Y 170.189,Z 274.697,A -85,B 0,C 180,E1 -24425.814,E2 -24425.814} C_VEL
LIN {X 0,Y 171.453,Z 255.425,A -85,B 0,C 180,E1 -24426.645,E2 -24426.645} C_VEL
LIN {X 0,Y 173.26,Z 224.791,A -85,B 0,C 180,E1 -24427.776,E2 -24427.776} C_VEL
LIN {X 0,Y 167.488,Z 212.887,A -85,B 0,C 180,E1 -24430.18,E2 -24430.18} C_VEL
LIN {X 0,Y 160.788,Z 201.291,A -85,B 0,C 180,E1 -24433.186,E2 -24433.186} C_VEL
LIN {X 0,Y 155.52,Z 193.38,A -85,B 0,C 180,E1 -24435.782,E2 -24435.782} C_VEL
LIN {X 0,Y 152.864,Z 189.614,A -85,B 0,C 180,E1 -24437.198,E2 -24437.198} C_VEL
LIN {X 0,Y 149.938,Z 185.529,A -85,B 0,C 180,E1 -24438.865,E2 -24438.865} C_VEL
LIN {X 0,Y 147.643,Z 182.712,A -85,B 0,C 180,E1 -24440.234,E2 -24440.234} C_VEL
LIN {X 0,Y 146.757,Z 181.01,A -85,B 0,C 180,E1 -24440.836,E2 -24440.836} C_VEL
LIN {X 0,Y 144.5,Z 179.017,A -85,B 0,C 180,E1 -24442.244,E2 -24442.244} C_VEL
LIN {X 0,Y 143.309,Z 176.677,A -85,B 0,C 180,E1 -24443.139,E2 -24443.139} C_VEL
LIN {X 0,Y 143.114,Z 175.654,A -85,B 0,C 180,E1 -24443.429,E2 -24443.429} C_VEL
LIN {X 0,Y 143.175,Z 175.64,A -85,B 0,C 180,E1 -24447.319,E2 -24447.319} C_VEL
LIN {X 0,Y 143.182,Z 175.638,A -85,B 0,C 180,E1 -24452.063,E2 -24452.063} C_VEL
LIN {X 0,Y 143.26,Z 175.626,A -85,B 0,C 180,E1 -24458.755,E2 -24458.755} C_VEL
LIN {X 0,Y 143.26,Z 175.632,A -85,B 0,C 180,E1 -24462.881,E2 -24462.881} C_VEL
LIN {X 0,Y 143.525,Z 175.602,A -85,B 0,C 180,E1 -24468.704,E2 -24468.704} C_VEL
LIN {X 0,Y 143.598,Z 175.551,A -85,B 0,C 180,E1 -24471.557,E2 -24471.557} C_VEL
LIN {X 0,Y 144.145,Z 175.53,A -85,B 0,C 180,E1 -24480,E2 -24480} C_VEL
LIN {X 0,Y 143.597,Z 175.595,A -85,B 0,C 180,E1 -24488.443,E2 -24488.443} C_VEL
LIN {X 0,Y 143.491,Z 175.606,A -85,B 0,C 180,E1 -24491.618,E2 -24491.618} C_VEL
LIN {X 0,Y 143.259,Z 175.639,A -85,B 0,C 180,E1 -24497.118,E2 -24497.118} C_VEL
LIN {X 0,Y 143.26,Z 175.64,A -85,B 0,C 180,E1 -24501.245,E2 -24501.245} C_VEL
LIN {X 0,Y 143.181,Z 175.652,A -85,B 0,C 180,E1 -24507.936,E2 -24507.936} C_VEL
LIN {X 0,Y 143.165,Z 175.658,A -85,B 0,C 180,E1 -24511.027,E2 -24511.027} C_VEL
LIN {X 0,Y 144.06,Z 178.329,A -85,B 0,C 180,E1 -24511.836,E2 -24511.836} C_VEL
LIN {X 0,Y 146.141,Z 180.598,A -85,B 0,C 180,E1 -24513.19,E2 -24513.19} C_VEL
LIN {X 0,Y 147.13,Z 181.532,A -85,B 0,C 180,E1 -24513.794,E2 -24513.794} C_VEL
LIN {X 0,Y 149.257,Z 184.818,A -85,B 0,C 180,E1 -24515.137,E2 -24515.137} C_VEL
LIN {X 0,Y 150.807,Z 186.574,A -85,B 0,C 180,E1 -24516.021,E2 -24516.021} C_VEL
LIN {X 0,Y 154.197,Z 191.801,A -85,B 0,C 180,E1 -24517.935,E2 -24517.935} C_VEL
LIN {X 0,Y 158.798,Z 199.969,A -85,B 0,C 180,E1 -24520.367,E2 -24520.367} C_VEL
LIN {X 0,Y 164.625,Z 211.948,A -85,B 0,C 180,E1 -24523.214,E2 -24523.214} C_VEL
LIN {X 0,Y 168.85,Z 222.247,A -85,B 0,C 180,E1 -24525.17,E2 -24525.17} C_VEL
LIN {X 0,Y 171.143,Z 228.862,A -85,B 0,C 180,E1 -24526.224,E2 -24526.224} C_VEL
LIN {X 0,Y 172.189,Z 243.992,A -85,B 0,C 180,E1 -24527.339,E2 -24527.339} C_VEL
LIN {X 0,Y 169.639,Z 284.51,A -85,B 0,C 180,E1 -24528.88,E2 -24528.88} C_VEL
LIN {X 0,Y 167.953,Z 297.689,A -85,B 0,C 180,E1 -24529.764,E2 -24529.764} C_VEL
LIN {X 0,Y 165.778,Z 309.239,A -85,B 0,C 180,E1 -24530.908,E2 -24530.908} C_VEL
LIN {X 0,Y 162.976,Z 320.804,A -85,B 0,C 180,E1 -24532.478,E2 -24532.478} C_VEL
LIN {X 0,Y 159.445,Z 332.648,A -85,B 0,C 180,E1 -24534.657,E2 -24534.657} C_VEL
LIN {X 0,Y 155.812,Z 343.26,A -85,B 0,C 180,E1 -24537.233,E2 -24537.233} C_VEL
LIN {X 0,Y 152.197,Z 352.825,A -85,B 0,C 180,E1 -24540.241,E2 -24540.241} C_VEL
LIN {X 0,Y 148.631,Z 361.822,A -85,B 0,C 180,E1 -24543.95,E2 -24543.95} C_VEL
LIN {X 0,Y 146.117,Z 368.326,A -85,B 0,C 180,E1 -24547.373,E2 -24547.373} C_VEL
LIN {X 0,Y 143.696,Z 374.485,A -85,B 0,C 180,E1 -24551.467,E2 -24551.467} C_VEL
LIN {X 0,Y 141.967,Z 379.367,A -85,B 0,C 180,E1 -24555.672,E2 -24555.672} C_VEL
LIN {X 0,Y 141.038,Z 383.122,A -85,B 0,C 180,E1 -24559.959,E2 -24559.959} C_VEL
LIN {X 0,Y 140.725,Z 384.92,A -85,B 0,C 180,E1 -24562.698,E2 -24562.698} C_VEL
LIN {X 0,Y 140.327,Z 385.827,A -85,B 0,C 180,E1 -24564.26,E2 -24564.26} C_VEL
LIN {X 0,Y 138.906,Z 386.85,A -85,B 0,C 180,E1 -24566.589,E2 -24566.589} C_VEL
LIN {X 0,Y 134.582,Z 388.039,A -85,B 0,C 180,E1 -24572.172,E2 -24572.172} C_VEL
LIN {X 0,Y 133.59,Z 388.145,A -85,B 0,C 180,E1 -24574.714,E2 -24574.714} C_VEL
LIN {X 0,Y 133.529,Z 388.09,A -85,B 0,C 180,E1 -24575.576,E2 -24575.576} C_VEL
LIN {X 0,Y 133.792,Z 387.73,A -85,B 0,C 180,E1 -24579.07,E2 -24579.07} C_VEL
LIN {X 0,Y 134.329,Z 386.985,A -85,B 0,C 180,E1 -24582.083,E2 -24582.083} C_VEL
LIN {X 0,Y 135.194,Z 385.825,A -85,B 0,C 180,E1 -24585.068,E2 -24585.068} C_VEL
LIN {X 0,Y 136.366,Z 384.234,A -85,B 0,C 180,E1 -24588.015,E2 -24588.015} C_VEL
LIN {X 0,Y 138.971,Z 381.075,A -85,B 0,C 180,E1 -24592.292,E2 -24592.292} C_VEL
LIN {X 0,Y 142.28,Z 376.871,A -85,B 0,C 180,E1 -24596.398,E2 -24596.398} C_VEL
LIN {X 0,Y 146.796,Z 370.487,A -85,B 0,C 180,E1 -24600.978,E2 -24600.978} C_VEL
LIN {X 0,Y 151.522,Z 363.565,A -85,B 0,C 180,E1 -24604.626,E2 -24604.626} C_VEL
LIN {X 0,Y 156.965,Z 354.923,A -85,B 0,C 180,E1 -24608.001,E2 -24608.001} C_VEL
LIN {X 0,Y 161.881,Z 346.081,A -85,B 0,C 180,E1 -24610.636,E2 -24610.636} C_VEL
LIN {X 0,Y 167.25,Z 335.214,A -85,B 0,C 180,E1 -24613.068,E2 -24613.068} C_VEL
LIN {X 0,Y 171.735,Z 324.262,A -85,B 0,C 180,E1 -24614.907,E2 -24614.907} C_VEL
LIN {X 0,Y 175.832,Z 311.998,A -85,B 0,C 180,E1 -24616.426,E2 -24616.426} C_VEL
LIN {X 0,Y 178.84,Z 300.415,A -85,B 0,C 180,E1 -24617.464,E2 -24617.464} C_VEL
LIN {X 0,Y 181.121,Z 287.714,A -85,B 0,C 180,E1 -24618.273,E2 -24618.273} C_VEL
LIN {X 0,Y 182.628,Z 272.646,A -85,B 0,C 180,E1 -24618.847,E2 -24618.847} C_VEL
LIN {X 0,Y 184.124,Z 251.818,A -85,B 0,C 180,E1 -24619.542,E2 -24619.542} C_VEL
LIN {X 0,Y 179.889,Z 240.479,A -85,B 0,C 180,E1 -24622.026,E2 -24622.026} C_VEL
LIN {X 0,Y 175.652,Z 230.919,A -85,B 0,C 180,E1 -24624.672,E2 -24624.672} C_VEL
LIN {X 0,Y 171.399,Z 222.277,A -85,B 0,C 180,E1 -24627.601,E2 -24627.601} C_VEL
LIN {X 0,Y 167.265,Z 214.616,A -85,B 0,C 180,E1 -24630.815,E2 -24630.815} C_VEL
LIN {X 0,Y 164.022,Z 209.134,A -85,B 0,C 180,E1 -24633.688,E2 -24633.688} C_VEL
LIN {X 0,Y 161.188,Z 204.914,A -85,B 0,C 180,E1 -24636.535,E2 -24636.535} C_VEL
LIN {X 0,Y 158.535,Z 201.754,A -85,B 0,C 180,E1 -24639.578,E2 -24639.578} C_VEL
LIN {X 0,Y 157.651,Z 200.121,A -85,B 0,C 180,E1 -24640.822,E2 -24640.822} C_VEL
LIN {X 0,Y 155.249,Z 197.994,A -85,B 0,C 180,E1 -24644.408,E2 -24644.408} C_VEL
LIN {X 0,Y 153.868,Z 195.244,A -85,B 0,C 180,E1 -24647.432,E2 -24647.432} C_VEL
LIN {X 0,Y 153.643,Z 194.689,A -85,B 0,C 180,E1 -24648.047,E2 -24648.047} C_VEL
LIN {X 0,Y 151.696,Z 193.134,A -85,B 0,C 180,E1 -24660,E2 -24660} C_VEL
LIN {X 0,Y 153.937,Z 194.863,A -85,B 0,C 180,E1 -24668.285,E2 -24668.285} C_VEL
LIN {X 0,Y 155.342,Z 198.037,A -85,B 0,C 180,E1 -24671.417,E2 -24671.417} C_VEL
LIN {X 0,Y 157.994,Z 200.523,A -85,B 0,C 180,E1 -24675.315,E2 -24675.315} C_VEL
LIN {X 0,Y 160.023,Z 203.796,A -85,B 0,C 180,E1 -24677.905,E2 -24677.905} C_VEL
LIN {X 0,Y 161.956,Z 205.925,A -85,B 0,C 180,E1 -24679.941,E2 -24679.941} C_VEL
LIN {X 0,Y 165.403,Z 210.72,A -85,B 0,C 180,E1 -24683.187,E2 -24683.187} C_VEL
LIN {X 0,Y 168.551,Z 215.234,A -85,B 0,C 180,E1 -24685.757,E2 -24685.757} C_VEL
LIN {X 0,Y 171.838,Z 220.212,A -85,B 0,C 180,E1 -24688.157,E2 -24688.157} C_VEL
LIN {X 0,Y 176.365,Z 227.494,A -85,B 0,C 180,E1 -24691.107,E2 -24691.107} C_VEL
LIN {X 0,Y 182.067,Z 237.711,A -85,B 0,C 180,E1 -24694.406,E2 -24694.406} C_VEL
LIN {X 0,Y 184.759,Z 243.185,A -85,B 0,C 180,E1 -24695.851,E2 -24695.851} C_VEL
LIN {X 0,Y 182.329,Z 274.004,A -85,B 0,C 180,E1 -24696.92,E2 -24696.92} C_VEL
LIN {X 0,Y 180.273,Z 287.442,A -85,B 0,C 180,E1 -24697.747,E2 -24697.747} C_VEL
LIN {X 0,Y 177.278,Z 300.294,A -85,B 0,C 180,E1 -24698.919,E2 -24698.919} C_VEL
LIN {X 0,Y 173.527,Z 312.48,A -85,B 0,C 180,E1 -24700.49,E2 -24700.49} C_VEL
LIN {X 0,Y 169.128,Z 323.965,A -85,B 0,C 180,E1 -24702.471,E2 -24702.471} C_VEL
LIN {X 0,Y 165.036,Z 332.957,A -85,B 0,C 180,E1 -24704.494,E2 -24704.494} C_VEL
LIN {X 0,Y 160.108,Z 342.157,A -85,B 0,C 180,E1 -24707.125,E2 -24707.125} C_VEL
LIN {X 0,Y 154.78,Z 351.081,A -85,B 0,C 180,E1 -24710.526,E2 -24710.526} C_VEL
LIN {X 0,Y 150.068,Z 358.235,A -85,B 0,C 180,E1 -24714.166,E2 -24714.166} C_VEL
LIN {X 0,Y 145.717,Z 363.915,A -85,B 0,C 180,E1 -24717.956,E2 -24717.956} C_VEL
LIN {X 0,Y 142.08,Z 368.367,A -85,B 0,C 180,E1 -24721.969,E2 -24721.969} C_VEL
LIN {X 0,Y 139.041,Z 371.734,A -85,B 0,C 180,E1 -24726.146,E2 -24726.146} C_VEL
LIN {X 0,Y 137.428,Z 373.394,A -85,B 0,C 180,E1 -24729.021,E2 -24729.021} C_VEL
LIN {X 0,Y 135.062,Z 375.516,A -85,B 0,C 180,E1 -24734.917,E2 -24734.917} C_VEL
LIN {X 0,Y 134.372,Z 375.954,A -85,B 0,C 180,E1 -24737.921,E2 -24737.921} C_VEL
LIN {X 0,Y 133.954,Z 375.988,A -85,B 0,C 180,E1 -24740.941,E2 -24740.941} C_VEL
LIN {X 0,Y 133.789,Z 375.063,A -85,B 0,C 180,E1 -24746.461,E2 -24746.461} C_VEL
LIN {X 0,Y 133.947,Z 373.789,A -85,B 0,C 180,E1 -24749.997,E2 -24749.997} C_VEL
LIN {X 0,Y 134.385,Z 372.232,A -85,B 0,C 180,E1 -24752.995,E2 -24752.995} C_VEL
LIN {X 0,Y 135.503,Z 369.12,A -85,B 0,C 180,E1 -24757.447,E2 -24757.447} C_VEL
LIN {X 0,Y 137.199,Z 364.966,A -85,B 0,C 180,E1 -24761.821,E2 -24761.821} C_VEL
LIN {X 0,Y 140.059,Z 358.641,A -85,B 0,C 180,E1 -24766.767,E2 -24766.767} C_VEL
LIN {X 0,Y 143.313,Z 351.549,A -85,B 0,C 180,E1 -24770.937,E2 -24770.937} C_VEL
LIN {X 0,Y 146.891,Z 343.112,A -85,B 0,C 180,E1 -24774.745,E2 -24774.745} C_VEL
LIN {X 0,Y 150.432,Z 334.264,A -85,B 0,C 180,E1 -24777.849,E2 -24777.849} C_VEL
LIN {X 0,Y 153.918,Z 324.544,A -85,B 0,C 180,E1 -24780.526,E2 -24780.526} C_VEL
LIN {X 0,Y 157.198,Z 313.862,A -85,B 0,C 180,E1 -24782.822,E2 -24782.822} C_VEL
LIN {X 0,Y 160.244,Z 301.879,A -85,B 0,C 180,E1 -24784.758,E2 -24784.758} C_VEL
LIN {X 0,Y 162.716,Z 289.375,A -85,B 0,C 180,E1 -24786.238,E2 -24786.238} C_VEL
LIN {X 0,Y 164.518,Z 276.57,A -85,B 0,C 180,E1 -24787.264,E2 -24787.264} C_VEL
LIN {X 0,Y 165.741,Z 260.251,A -85,B 0,C 180,E1 -24788.026,E2 -24788.026} C_VEL
LIN {X 0,Y 167.793,Z 227.1,A -85,B 0,C 180,E1 -24789.272,E2 -24789.272} C_VEL
LIN {X 0,Y 162.65,Z 216.498,A -85,B 0,C 180,E1 -24791.578,E2 -24791.578} C_VEL
LIN {X 0,Y 156.894,Z 206.312,A -85,B 0,C 180,E1 -24794.352,E2 -24794.352} C_VEL
LIN {X 0,Y 152.037,Z 198.797,A -85,B 0,C 180,E1 -24796.909,E2 -24796.909} C_VEL
LIN {X 0,Y 148.548,Z 193.824,A -85,B 0,C 180,E1 -24798.91,E2 -24798.91} C_VEL
LIN {X 0,Y 146.771,Z 191.269,A -85,B 0,C 180,E1 -24800.004,E2 -24800.004} C_VEL
LIN {X 0,Y 144.243,Z 187.806,A -85,B 0,C 180,E1 -24801.644,E2 -24801.644} C_VEL
LIN {X 0,Y 143.503,Z 186.834,A -85,B 0,C 180,E1 -24802.144,E2 -24802.144} C_VEL
LIN {X 0,Y 141.179,Z 184.136,A -85,B 0,C 180,E1 -24803.761,E2 -24803.761} C_VEL
LIN {X 0,Y 139.957,Z 182.032,A -85,B 0,C 180,E1 -24804.726,E2 -24804.726} C_VEL
LIN {X 0,Y 137.667,Z 180.187,A -85,B 0,C 180,E1 -24806.446,E2 -24806.446} C_VEL
LIN {X 0,Y 136.343,Z 177.581,A -85,B 0,C 180,E1 -24807.669,E2 -24807.669} C_VEL
LIN {X 0,Y 136.081,Z 176.525,A -85,B 0,C 180,E1 -24808.037,E2 -24808.037} C_VEL
LIN {X 0,Y 136.137,Z 176.515,A -85,B 0,C 180,E1 -24812.314,E2 -24812.314} C_VEL
LIN {X 0,Y 136.226,Z 176.502,A -85,B 0,C 180,E1 -24818.83,E2 -24818.83} C_VEL
LIN {X 0,Y 136.225,Z 176.501,A -85,B 0,C 180,E1 -24825.051,E2 -24825.051} C_VEL
LIN {X 0,Y 136.418,Z 176.491,A -85,B 0,C 180,E1 -24828.177,E2 -24828.177} C_VEL
LIN {X 0,Y 136.527,Z 176.435,A -85,B 0,C 180,E1 -24831.116,E2 -24831.116} C_VEL
LIN {X 0,Y 137.102,Z 176.407,A -85,B 0,C 180,E1 -24840,E2 -24840} C_VEL
LIN {X 0,Y 136.527,Z 176.478,A -85,B 0,C 180,E1 -24848.884,E2 -24848.884} C_VEL
LIN {X 0,Y 136.406,Z 176.488,A -85,B 0,C 180,E1 -24851.893,E2 -24851.893} C_VEL
LIN {X 0,Y 136.18,Z 176.526,A -85,B 0,C 180,E1 -24858.038,E2 -24858.038} C_VEL
LIN {X 0,Y 136.182,Z 176.523,A -85,B 0,C 180,E1 -24861.74,E2 -24861.74} C_VEL
LIN {X 0,Y 136.109,Z 176.603,A -85,B 0,C 180,E1 -24866.446,E2 -24866.446} C_VEL
LIN {X 0,Y 137.018,Z 179.223,A -85,B 0,C 180,E1 -24867.389,E2 -24867.389} C_VEL
LIN {X 0,Y 139.259,Z 181.618,A -85,B 0,C 180,E1 -24869.172,E2 -24869.172} C_VEL
LIN {X 0,Y 140.349,Z 182.435,A -85,B 0,C 180,E1 -24869.955,E2 -24869.955} C_VEL
LIN {X 0,Y 142.192,Z 185.502,A -85,B 0,C 180,E1 -24871.367,E2 -24871.367} C_VEL
LIN {X 0,Y 144.3,Z 187.737,A -85,B 0,C 180,E1 -24872.772,E2 -24872.772} C_VEL
LIN {X 0,Y 146.77,Z 191.194,A -85,B 0,C 180,E1 -24874.379,E2 -24874.379} C_VEL
LIN {X 0,Y 148.275,Z 193.315,A -85,B 0,C 180,E1 -24875.306,E2 -24875.306} C_VEL
LIN {X 0,Y 150.608,Z 197.02,A -85,B 0,C 180,E1 -24876.702,E2 -24876.702} C_VEL
LIN {X 0,Y 154.877,Z 204.873,A -85,B 0,C 180,E1 -24879.127,E2 -24879.127} C_VEL
LIN {X 0,Y 160.379,Z 216.55,A -85,B 0,C 180,E1 -24882.013,E2 -24882.013} C_VEL
LIN {X 0,Y 164.595,Z 227.275,A -85,B 0,C 180,E1 -24884.11,E2 -24884.11} C_VEL
LIN {X 0,Y 165.965,Z 231.482,A -85,B 0,C 180,E1 -24884.796,E2 -24884.796} C_VEL
LIN {X 0,Y 166.791,Z 244.127,A -85,B 0,C 180,E1 -24885.773,E2 -24885.773} C_VEL
LIN {X 0,Y 164.236,Z 283.554,A -85,B 0,C 180,E1 -24887.294,E2 -24887.294} C_VEL
LIN {X 0,Y 162.537,Z 296.652,A -85,B 0,C 180,E1 -24888.169,E2 -24888.169} C_VEL
LIN {X 0,Y 160.344,Z 308.172,A -85,B 0,C 180,E1 -24889.313,E2 -24889.313} C_VEL
LIN {X 0,Y 157.403,Z 319.9,A -85,B 0,C 180,E1 -24890.903,E2 -24890.903} C_VEL
LIN {X 0,Y 154.119,Z 330.582,A -85,B 0,C 180,E1 -24892.831,E2 -24892.831} C_VEL
LIN {X 0,Y 150.309,Z 341.509,A -85,B 0,C 180,E1 -24895.467,E2 -24895.467} C_VEL
LIN {X 0,Y 146.033,Z 352.211,A -85,B 0,C 180,E1 -24898.848,E2 -24898.848} C_VEL
LIN {X 0,Y 142.662,Z 360.39,A -85,B 0,C 180,E1 -24902.258,E2 -24902.258} C_VEL
LIN {X 0,Y 139.578,Z 367.819,A -85,B 0,C 180,E1 -24906.249,E2 -24906.249} C_VEL
LIN {X 0,Y 136.962,Z 374.013,A -85,B 0,C 180,E1 -24910.52,E2 -24910.52} C_VEL
LIN {X 0,Y 135.035,Z 378.923,A -85,B 0,C 180,E1 -24914.919,E2 -24914.919} C_VEL
LIN {X 0,Y 134.023,Z 382.71,A -85,B 0,C 180,E1 -24919.427,E2 -24919.427} C_VEL
LIN {X 0,Y 133.583,Z 385.458,A -85,B 0,C 180,E1 -24923.963,E2 -24923.963} C_VEL
LIN {X 0,Y 133.643,Z 387.005,A -85,B 0,C 180,E1 -24927.66,E2 -24927.66} C_VEL
LIN {X 0,Y 133.776,Z 387.645,A -85,B 0,C 180,E1 -24930.003,E2 -24930.003} C_VEL
LIN {X 0,Y 133.601,Z 388.075,A -85,B 0,C 180,E1 -24933.018,E2 -24933.018} C_VEL
LIN {X 0,Y 133.529,Z 388.09,A -85,B 0,C 180,E1 -24935.576,E2 -24935.576} C_VEL
LIN {X 0,Y 132.999,Z 387.953,A -85,B 0,C 180,E1 -24938.107,E2 -24938.107} C_VEL
LIN {X 0,Y 130.753,Z 387.075,A -85,B 0,C 180,E1 -24942.297,E2 -24942.297} C_VEL
LIN {X 0,Y 129.163,Z 385.361,A -85,B 0,C 180,E1 -24946.563,E2 -24946.563} C_VEL
LIN {X 0,Y 129.662,Z 383.912,A -85,B 0,C 180,E1 -24949.097,E2 -24949.097} C_VEL
LIN {X 0,Y 132.406,Z 380.853,A -85,B 0,C 180,E1 -24953.462,E2 -24953.462} C_VEL
LIN {X 0,Y 136.671,Z 375.675,A -85,B 0,C 180,E1 -24958.599,E2 -24958.599} C_VEL
LIN {X 0,Y 141.487,Z 369.305,A -85,B 0,C 180,E1 -24963.123,E2 -24963.123} C_VEL
LIN {X 0,Y 146.646,Z 362.134,A -85,B 0,C 180,E1 -24966.805,E2 -24966.805} C_VEL
LIN {X 0,Y 152.433,Z 353.237,A -85,B 0,C 180,E1 -24970.204,E2 -24970.204} C_VEL
LIN {X 0,Y 157.681,Z 344.126,A -85,B 0,C 180,E1 -24972.823,E2 -24972.823} C_VEL
LIN {X 0,Y 162.691,Z 334.056,A -85,B 0,C 180,E1 -24975.024,E2 -24975.024} C_VEL
LIN {X 0,Y 167.413,Z 322.878,A -85,B 0,C 180,E1 -24976.839,E2 -24976.839} C_VEL
LIN {X 0,Y 171.632,Z 310.345,A -85,B 0,C 180,E1 -24978.36,E2 -24978.36} C_VEL
LIN {X 0,Y 174.891,Z 297.479,A -85,B 0,C 180,E1 -24979.444,E2 -24979.444} C_VEL
LIN {X 0,Y 177.185,Z 283.785,A -85,B 0,C 180,E1 -24980.218,E2 -24980.218} C_VEL
LIN {X 0,Y 179.61,Z 254.194,A -85,B 0,C 180,E1 -24981.239,E2 -24981.239} C_VEL
LIN {X 0,Y 175.729,Z 243.559,A -85,B 0,C 180,E1 -24983.722,E2 -24983.722} C_VEL
LIN {X 0,Y 171.345,Z 233.388,A -85,B 0,C 180,E1 -24986.739,E2 -24986.739} C_VEL
LIN {X 0,Y 167.237,Z 224.978,A -85,B 0,C 180,E1 -24989.89,E2 -24989.89} C_VEL
LIN {X 0,Y 164.479,Z 219.874,A -85,B 0,C 180,E1 -24992.253,E2 -24992.253} C_VEL
LIN {X 0,Y 162.008,Z 215.403,A -85,B 0,C 180,E1 -24994.624,E2 -24994.624} C_VEL
LIN {X 0,Y 159.41,Z 211.434,A -85,B 0,C 180,E1 -24997.394,E2 -24997.394} C_VEL
LIN {X 0,Y 156.704,Z 207.829,A -85,B 0,C 180,E1 -25000.769,E2 -25000.769} C_VEL
LIN {X 0,Y 156.121,Z 206.863,A -85,B 0,C 180,E1 -25001.633,E2 -25001.633} C_VEL
LIN {X 0,Y 153.689,Z 204.341,A -85,B 0,C 180,E1 -25005.645,E2 -25005.645} C_VEL
LIN {X 0,Y 152.5,Z 201.636,A -85,B 0,C 180,E1 -25008.668,E2 -25008.668} C_VEL
LIN {X 0,Y 150.829,Z 200.183,A -85,B 0,C 180,E1 -25020,E2 -25020} C_VEL
LIN {X 0,Y 152.754,Z 201.717,A -85,B 0,C 180,E1 -25027.601,E2 -25027.601} C_VEL
LIN {X 0,Y 154.114,Z 204.855,A -85,B 0,C 180,E1 -25030.843,E2 -25030.843} C_VEL
LIN {X 0,Y 156.534,Z 207.352,A -85,B 0,C 180,E1 -25034.629,E2 -25034.629} C_VEL
LIN {X 0,Y 158.851,Z 210.909,A -85,B 0,C 180,E1 -25037.667,E2 -25037.667} C_VEL
LIN {X 0,Y 160.19,Z 212.458,A -85,B 0,C 180,E1 -25039.139,E2 -25039.139} C_VEL
LIN {X 0,Y 163.632,Z 217.473,A -85,B 0,C 180,E1 -25042.553,E2 -25042.553} C_VEL
LIN {X 0,Y 166.694,Z 222.025,A -85,B 0,C 180,E1 -25045.162,E2 -25045.162} C_VEL
LIN {X 0,Y 171.131,Z 229.096,A -85,B 0,C 180,E1 -25048.474,E2 -25048.474} C_VEL
LIN {X 0,Y 175.724,Z 237.217,A -85,B 0,C 180,E1 -25051.496,E2 -25051.496} C_VEL
LIN {X 0,Y 180.247,Z 246.097,A -85,B 0,C 180,E1 -25054.177,E2 -25054.177} C_VEL
LIN {X 0,Y 177.912,Z 274.268,A -85,B 0,C 180,E1 -25055.158,E2 -25055.158} C_VEL
LIN {X 0,Y 175.772,Z 287.796,A -85,B 0,C 180,E1 -25055.995,E2 -25055.995} C_VEL
LIN {X 0,Y 172.901,Z 299.876,A -85,B 0,C 180,E1 -25057.086,E2 -25057.086} C_VEL
LIN {X 0,Y 169.203,Z 311.535,A -85,B 0,C 180,E1 -25058.539,E2 -25058.539} C_VEL
LIN {X 0,Y 164.971,Z 322.523,A -85,B 0,C 180,E1 -25060.401,E2 -25060.401} C_VEL
LIN {X 0,Y 160.118,Z 332.897,A -85,B 0,C 180,E1 -25062.673,E2 -25062.673} C_VEL
LIN {X 0,Y 154.954,Z 342.181,A -85,B 0,C 180,E1 -25065.329,E2 -25065.329} C_VEL
LIN {X 0,Y 149.317,Z 351.155,A -85,B 0,C 180,E1 -25068.778,E2 -25068.778} C_VEL
LIN {X 0,Y 144.326,Z 358.358,A -85,B 0,C 180,E1 -25072.503,E2 -25072.503} C_VEL
LIN {X 0,Y 139.692,Z 364.09,A -85,B 0,C 180,E1 -25076.396,E2 -25076.396} C_VEL
LIN {X 0,Y 135.805,Z 368.577,A -85,B 0,C 180,E1 -25080.55,E2 -25080.55} C_VEL
LIN {X 0,Y 132.527,Z 371.975,A -85,B 0,C 180,E1 -25084.894,E2 -25084.894} C_VEL
LIN {X 0,Y 130.765,Z 373.653,A -85,B 0,C 180,E1 -25087.898,E2 -25087.898} C_VEL
LIN {X 0,Y 128.153,Z 375.806,A -85,B 0,C 180,E1 -25094.083,E2 -25094.083} C_VEL
LIN {X 0,Y 127.384,Z 376.273,A -85,B 0,C 180,E1 -25097.248,E2 -25097.248} C_VEL
LIN {X 0,Y 126.704,Z 375.99,A -85,B 0,C 180,E1 -25103.628,E2 -25103.628} C_VEL
LIN {X 0,Y 126.701,Z 375.283,A -85,B 0,C 180,E1 -25106.817,E2 -25106.817} C_VEL
LIN {X 0,Y 126.851,Z 374.179,A -85,B 0,C 180,E1 -25109.997,E2 -25109.997} C_VEL
LIN {X 0,Y 127.314,Z 372.637,A -85,B 0,C 180,E1 -25113.162,E2 -25113.162} C_VEL
LIN {X 0,Y 128.504,Z 369.556,A -85,B 0,C 180,E1 -25117.855,E2 -25117.855} C_VEL
LIN {X 0,Y 130.299,Z 365.435,A -85,B 0,C 180,E1 -25122.456,E2 -25122.456} C_VEL
LIN {X 0,Y 133.319,Z 359.147,A -85,B 0,C 180,E1 -25127.642,E2 -25127.642} C_VEL
LIN {X 0,Y 136.967,Z 351.622,A -85,B 0,C 180,E1 -25132.25,E2 -25132.25} C_VEL
LIN {X 0,Y 140.435,Z 343.893,A -85,B 0,C 180,E1 -25135.886,E2 -25135.886} C_VEL
LIN {X 0,Y 144.215,Z 334.945,A -85,B 0,C 180,E1 -25139.162,E2 -25139.162} C_VEL
LIN {X 0,Y 148.289,Z 324.127,A -85,B 0,C 180,E1 -25142.217,E2 -25142.217} C_VEL
LIN {X 0,Y 151.75,Z 313.197,A -85,B 0,C 180,E1 -25144.561,E2 -25144.561} C_VEL
LIN {X 0,Y 154.98,Z 300.954,A -85,B 0,C 180,E1 -25146.522,E2 -25146.522} C_VEL
LIN {X 0,Y 157.335,Z 289.357,A -85,B 0,C 180,E1 -25147.89,E2 -25147.89} C_VEL
LIN {X 0,Y 159.154,Z 276.857,A -85,B 0,C 180,E1 -25148.9,E2 -25148.9} C_VEL
LIN {X 0,Y 160.395,Z 261.303,A -85,B 0,C 180,E1 -25149.643,E2 -25149.643} C_VEL
LIN {X 0,Y 162.459,Z 229.491,A -85,B 0,C 180,E1 -25150.859,E2 -25150.859} C_VEL
LIN {X 0,Y 157.858,Z 219.914,A -85,B 0,C 180,E1 -25153.094,E2 -25153.094} C_VEL
LIN {X 0,Y 152.822,Z 210.895,A -85,B 0,C 180,E1 -25155.711,E2 -25155.711} C_VEL
LIN {X 0,Y 148.014,Z 203.275,A -85,B 0,C 180,E1 -25158.448,E2 -25158.448} C_VEL
LIN {X 0,Y 143.675,Z 196.973,A -85,B 0,C 180,E1 -25161.19,E2 -25161.19} C_VEL
LIN {X 0,Y 140.511,Z 192.644,A -85,B 0,C 180,E1 -25163.401,E2 -25163.401} C_VEL
LIN {X 0,Y 137.975,Z 189.209,A -85,B 0,C 180,E1 -25165.345,E2 -25165.345} C_VEL
LIN {X 0,Y 137.162,Z 188.174,A -85,B 0,C 180,E1 -25166,E2 -25166} C_VEL
LIN {X 0,Y 134.752,Z 185.586,A -85,B 0,C 180,E1 -25168.019,E2 -25168.019} C_VEL
LIN {X 0,Y 133.442,Z 183.138,A -85,B 0,C 180,E1 -25169.321,E2 -25169.321} C_VEL
LIN {X 0,Y 130.941,Z 181.395,A -85,B 0,C 180,E1 -25171.691,E2 -25171.691} C_VEL
LIN {X 0,Y 129.404,Z 178.969,A -85,B 0,C 180,E1 -25173.489,E2 -25173.489} C_VEL
LIN {X 0,Y 129.02,Z 177.407,A -85,B 0,C 180,E1 -25174.165,E2 -25174.165} C_VEL
LIN {X 0,Y 129.099,Z 177.39,A -85,B 0,C 180,E1 -25177.729,E2 -25177.729} C_VEL
LIN {X 0,Y 129.15,Z 177.382,A -85,B 0,C 180,E1 -25184.211,E2 -25184.211} C_VEL
LIN {X 0,Y 129.337,Z 177.373,A -85,B 0,C 180,E1 -25187.969,E2 -25187.969} C_VEL
LIN {X 0,Y 129.453,Z 177.321,A -85,B 0,C 180,E1 -25190.626,E2 -25190.626} C_VEL
LIN {X 0,Y 130.057,Z 177.285,A -85,B 0,C 180,E1 -25200,E2 -25200} C_VEL
LIN {X 0,Y 129.453,Z 177.362,A -85,B 0,C 180,E1 -25209.373,E2 -25209.373} C_VEL
LIN {X 0,Y 129.29,Z 177.376,A -85,B 0,C 180,E1 -25212.558,E2 -25212.558} C_VEL
LIN {X 0,Y 129.113,Z 177.402,A -85,B 0,C 180,E1 -25219.889,E2 -25219.889} C_VEL
LIN {X 0,Y 129.14,Z 177.397,A -85,B 0,C 180,E1 -25220.404,E2 -25220.404} C_VEL
LIN {X 0,Y 129.992,Z 179.968,A -85,B 0,C 180,E1 -25221.621,E2 -25221.621} C_VEL
LIN {X 0,Y 131.8,Z 182.2,A -85,B 0,C 180,E1 -25223.573,E2 -25223.573} C_VEL
LIN {X 0,Y 133.672,Z 183.41,A -85,B 0,C 180,E1 -25225.289,E2 -25225.289} C_VEL
LIN {X 0,Y 135.358,Z 186.387,A -85,B 0,C 180,E1 -25226.916,E2 -25226.916} C_VEL
LIN {X 0,Y 137.775,Z 188.81,A -85,B 0,C 180,E1 -25228.874,E2 -25228.874} C_VEL
LIN {X 0,Y 140.168,Z 192.236,A -85,B 0,C 180,E1 -25230.743,E2 -25230.743} C_VEL
LIN {X 0,Y 141.602,Z 193.939,A -85,B 0,C 180,E1 -25231.76,E2 -25231.76} C_VEL
LIN {X 0,Y 145.123,Z 198.952,A -85,B 0,C 180,E1 -25234.143,E2 -25234.143} C_VEL
LIN {X 0,Y 147.135,Z 202.264,A -85,B 0,C 180,E1 -25235.433,E2 -25235.433} C_VEL
LIN {X 0,Y 151.25,Z 210.199,A -85,B 0,C 180,E1 -25237.948,E2 -25237.948} C_VEL
LIN {X 0,Y 155.859,Z 220.344,A -85,B 0,C 180,E1 -25240.558,E2 -25240.558} C_VEL
LIN {X 0,Y 159.519,Z 229.844,A -85,B 0,C 180,E1 -25242.532,E2 -25242.532} C_VEL
LIN {X 0,Y 160.879,Z 233.925,A -85,B 0,C 180,E1 -25243.26,E2 -25243.26} C_VEL
LIN {X 0,Y 161.496,Z 245.503,A -85,B 0,C 180,E1 -25244.168,E2 -25244.168} C_VEL
LIN {X 0,Y 158.883,Z 283.296,A -85,B 0,C 180,E1 -25245.638,E2 -25245.638} C_VEL
LIN {X 0,Y 157.137,Z 296.195,A -85,B 0,C 180,E1 -25246.509,E2 -25246.509} C_VEL
LIN {X 0,Y 154.761,Z 308.235,A -85,B 0,C 180,E1 -25247.731,E2 -25247.731} C_VEL
LIN {X 0,Y 151.449,Z 320.731,A -85,B 0,C 180,E1 -25249.487,E2 -25249.487} C_VEL
LIN {X 0,Y 147.558,Z 332.44,A -85,B 0,C 180,E1 -25251.748,E2 -25251.748} C_VEL
LIN {X 0,Y 143.608,Z 342.981,A -85,B 0,C 180,E1 -25254.473,E2 -25254.473} C_VEL
LIN {X 0,Y 139.962,Z 351.589,A -85,B 0,C 180,E1 -25257.334,E2 -25257.334} C_VEL
LIN {X 0,Y 136.499,Z 359.544,A -85,B 0,C 180,E1 -25260.722,E2 -25260.722} C_VEL
LIN {X 0,Y 133.606,Z 366.279,A -85,B 0,C 180,E1 -25264.375,E2 -25264.375} C_VEL
LIN {X 0,Y 131.115,Z 371.615,A -85,B 0,C 180,E1 -25267.966,E2 -25267.966} C_VEL
LIN {X 0,Y 128.728,Z 376.972,A -85,B 0,C 180,E1 -25272.529,E2 -25272.529} C_VEL
LIN {X 0,Y 127.304,Z 381.154,A -85,B 0,C 180,E1 -25277.246,E2 -25277.246} C_VEL
LIN {X 0,Y 126.773,Z 383.355,A -85,B 0,C 180,E1 -25280.43,E2 -25280.43} C_VEL
LIN {X 0,Y 126.519,Z 385.075,A -85,B 0,C 180,E1 -25283.624,E2 -25283.624} C_VEL
LIN {X 0,Y 126.577,Z 386.796,A -85,B 0,C 180,E1 -25288.053,E2 -25288.053} C_VEL
LIN {X 0,Y 126.574,Z 387.594,A -85,B 0,C 180,E1 -25291.914,E2 -25291.914} C_VEL
LIN {X 0,Y 126.462,Z 387.775,A -85,B 0,C 180,E1 -25296.384,E2 -25296.384} C_VEL
LIN {X 0,Y 127.366,Z 386.692,A -85,B 0,C 180,E1 -25302.754,E2 -25302.754} C_VEL
LIN {X 0,Y 128.301,Z 385.558,A -85,B 0,C 180,E1 -25305.898,E2 -25305.898} C_VEL
LIN {X 0,Y 129.662,Z 383.912,A -85,B 0,C 180,E1 -25309.097,E2 -25309.097} C_VEL
LIN {X 0,Y 130.416,Z 382.372,A -85,B 0,C 180,E1 -25311.578,E2 -25311.578} C_VEL
LIN {X 0,Y 130.357,Z 379.343,A -85,B 0,C 180,E1 -25315.739,E2 -25315.739} C_VEL
LIN {X 0,Y 130.843,Z 375.705,A -85,B 0,C 180,E1 -25319.799,E2 -25319.799} C_VEL
LIN {X 0,Y 132.399,Z 373.117,A -85,B 0,C 180,E1 -25322.022,E2 -25322.022} C_VEL
LIN {X 0,Y 137.312,Z 366.928,A -85,B 0,C 180,E1 -25326.061,E2 -25326.061} C_VEL
LIN {X 0,Y 142.985,Z 359.313,A -85,B 0,C 180,E1 -25329.718,E2 -25329.718} C_VEL
LIN {X 0,Y 148.16,Z 351.541,A -85,B 0,C 180,E1 -25332.531,E2 -25332.531} C_VEL
LIN {X 0,Y 153.672,Z 342.069,A -85,B 0,C 180,E1 -25335.146,E2 -25335.146} C_VEL
LIN {X 0,Y 158.951,Z 331.578,A -85,B 0,C 180,E1 -25337.316,E2 -25337.316} C_VEL
LIN {X 0,Y 163.921,Z 319.911,A -85,B 0,C 180,E1 -25339.085,E2 -25339.085} C_VEL
LIN {X 0,Y 168.021,Z 307.466,A -85,B 0,C 180,E1 -25340.465,E2 -25340.465} C_VEL
LIN {X 0,Y 171.232,Z 293.981,A -85,B 0,C 180,E1 -25341.544,E2 -25341.544} C_VEL
LIN {X 0,Y 173.246,Z 281.236,A -85,B 0,C 180,E1 -25342.176,E2 -25342.176} C_VEL
LIN {X 0,Y 175.258,Z 256.623,A -85,B 0,C 180,E1 -25343.022,E2 -25343.022} C_VEL
LIN {X 0,Y 171.846,Z 247.077,A -85,B 0,C 180,E1 -25345.405,E2 -25345.405} C_VEL
LIN {X 0,Y 168.084,Z 238.083,A -85,B 0,C 180,E1 -25348.226,E2 -25348.226} C_VEL
LIN {X 0,Y 164.525,Z 230.386,A -85,B 0,C 180,E1 -25351.201,E2 -25351.201} C_VEL
LIN {X 0,Y 161.915,Z 225.304,A -85,B 0,C 180,E1 -25353.631,E2 -25353.631} C_VEL
LIN {X 0,Y 159.756,Z 221.233,A -85,B 0,C 180,E1 -25355.882,E2 -25355.882} C_VEL
LIN {X 0,Y 157.687,Z 217.946,A -85,B 0,C 180,E1 -25358.255,E2 -25358.255} C_VEL
LIN {X 0,Y 155.034,Z 214.079,A -85,B 0,C 180,E1 -25361.841,E2 -25361.841} C_VEL
LIN {X 0,Y 152.124,Z 210.423,A -85,B 0,C 180,E1 -25367.126,E2 -25367.126} C_VEL
LIN {X 0,Y 151.375,Z 208.582,A -85,B 0,C 180,E1 -25369.298,E2 -25369.298} C_VEL
LIN {X 0,Y 149.962,Z 207.231,A -85,B 0,C 180,E1 -25380,E2 -25380} C_VEL
LIN {X 0,Y 151.67,Z 208.809,A -85,B 0,C 180,E1 -25387.154,E2 -25387.154} C_VEL
LIN {X 0,Y 153.151,Z 212.014,A -85,B 0,C 180,E1 -25390.745,E2 -25390.745} C_VEL
LIN {X 0,Y 155.105,Z 214.12,A -85,B 0,C 180,E1 -25393.929,E2 -25393.929} C_VEL
LIN {X 0,Y 157.539,Z 217.827,A -85,B 0,C 180,E1 -25397.254,E2 -25397.254} C_VEL
LIN {X 0,Y 158.6,Z 219.248,A -85,B 0,C 180,E1 -25398.489,E2 -25398.489} C_VEL
LIN {X 0,Y 161.678,Z 223.878,A -85,B 0,C 180,E1 -25401.705,E2 -25401.705} C_VEL
LIN {X 0,Y 165.547,Z 229.872,A -85,B 0,C 180,E1 -25405.121,E2 -25405.121} C_VEL
LIN {X 0,Y 170.066,Z 237.767,A -85,B 0,C 180,E1 -25408.573,E2 -25408.573} C_VEL
LIN {X 0,Y 174.623,Z 246.482,A -85,B 0,C 180,E1 -25411.628,E2 -25411.628} C_VEL
LIN {X 0,Y 175.897,Z 249.085,A -85,B 0,C 180,E1 -25412.424,E2 -25412.424} C_VEL
LIN {X 0,Y 173.599,Z 275.175,A -85,B 0,C 180,E1 -25413.343,E2 -25413.343} C_VEL
LIN {X 0,Y 171.326,Z 288.731,A -85,B 0,C 180,E1 -25414.19,E2 -25414.19} C_VEL
LIN {X 0,Y 168.387,Z 300.477,A -85,B 0,C 180,E1 -25415.263,E2 -25415.263} C_VEL
LIN {X 0,Y 164.472,Z 312.28,A -85,B 0,C 180,E1 -25416.744,E2 -25416.744} C_VEL
LIN {X 0,Y 159.855,Z 323.669,A -85,B 0,C 180,E1 -25418.702,E2 -25418.702} C_VEL
LIN {X 0,Y 154.81,Z 333.871,A -85,B 0,C 180,E1 -25420.995,E2 -25420.995} C_VEL
LIN {X 0,Y 148.903,Z 343.835,A -85,B 0,C 180,E1 -25423.961,E2 -25423.961} C_VEL
LIN {X 0,Y 143.206,Z 352.365,A -85,B 0,C 180,E1 -25427.405,E2 -25427.405} C_VEL
LIN {X 0,Y 137.846,Z 359.529,A -85,B 0,C 180,E1 -25431.348,E2 -25431.348} C_VEL
LIN {X 0,Y 132.302,Z 365.873,A -85,B 0,C 180,E1 -25436.096,E2 -25436.096} C_VEL
LIN {X 0,Y 128.351,Z 370.021,A -85,B 0,C 180,E1 -25440.472,E2 -25440.472} C_VEL
LIN {X 0,Y 126.08,Z 372.212,A -85,B 0,C 180,E1 -25443.514,E2 -25443.514} C_VEL
LIN {X 0,Y 124.147,Z 373.913,A -85,B 0,C 180,E1 -25446.652,E2 -25446.652} C_VEL
LIN {X 0,Y 121.279,Z 376.095,A -85,B 0,C 180,E1 -25453.154,E2 -25453.154} C_VEL
LIN {X 0,Y 120.426,Z 376.589,A -85,B 0,C 180,E1 -25456.497,E2 -25456.497} C_VEL
LIN {X 0,Y 119.892,Z 376.653,A -85,B 0,C 180,E1 -25459.868,E2 -25459.868} C_VEL
LIN {X 0,Y 119.638,Z 376.336,A -85,B 0,C 180,E1 -25463.25,E2 -25463.25} C_VEL
LIN {X 0,Y 119.61,Z 375.474,A -85,B 0,C 180,E1 -25467.3,E2 -25467.3} C_VEL
LIN {X 0,Y 120.245,Z 373.042,A -85,B 0,C 180,E1 -25473.348,E2 -25473.348} C_VEL
LIN {X 0,Y 121.514,Z 369.991,A -85,B 0,C 180,E1 -25478.311,E2 -25478.311} C_VEL
LIN {X 0,Y 123.417,Z 365.905,A -85,B 0,C 180,E1 -25483.163,E2 -25483.163} C_VEL
LIN {X 0,Y 126.614,Z 359.654,A -85,B 0,C 180,E1 -25488.609,E2 -25488.609} C_VEL
LIN {X 0,Y 130.089,Z 352.852,A -85,B 0,C 180,E1 -25493.055,E2 -25493.055} C_VEL
LIN {X 0,Y 134.185,Z 344.352,A -85,B 0,C 180,E1 -25497.273,E2 -25497.273} C_VEL
LIN {X 0,Y 138.09,Z 335.625,A -85,B 0,C 180,E1 -25500.59,E2 -25500.59} C_VEL
LIN {X 0,Y 142.378,Z 324.884,A -85,B 0,C 180,E1 -25503.729,E2 -25503.729} C_VEL
LIN {X 0,Y 146.001,Z 314.098,A -85,B 0,C 180,E1 -25506.13,E2 -25506.13} C_VEL
LIN {X 0,Y 149.373,Z 302.004,A -85,B 0,C 180,E1 -25508.132,E2 -25508.132} C_VEL
LIN {X 0,Y 152.101,Z 289.336,A -85,B 0,C 180,E1 -25509.656,E2 -25509.656} C_VEL
LIN {X 0,Y 154.045,Z 276.285,A -85,B 0,C 180,E1 -25510.694,E2 -25510.694} C_VEL
LIN {X 0,Y 155.378,Z 259.147,A -85,B 0,C 180,E1 -25511.504,E2 -25511.504} C_VEL
LIN {X 0,Y 157.244,Z 231.852,A -85,B 0,C 180,E1 -25512.558,E2 -25512.558} C_VEL
LIN {X 0,Y 152.341,Z 221.741,A -85,B 0,C 180,E1 -25515.161,E2 -25515.161} C_VEL
LIN {X 0,Y 147,Z 212.313,A -85,B 0,C 180,E1 -25518.249,E2 -25518.249} C_VEL
LIN {X 0,Y 141.019,Z 203.075,A -85,B 0,C 180,E1 -25522.172,E2 -25522.172} C_VEL
LIN {X 0,Y 137.584,Z 198.381,A -85,B 0,C 180,E1 -25524.721,E2 -25524.721} C_VEL
LIN {X 0,Y 134.695,Z 194.374,A -85,B 0,C 180,E1 -25527.13,E2 -25527.13} C_VEL
LIN {X 0,Y 132.105,Z 191.214,A -85,B 0,C 180,E1 -25529.499,E2 -25529.499} C_VEL
LIN {X 0,Y 131.198,Z 189.642,A -85,B 0,C 180,E1 -25530.453,E2 -25530.453} C_VEL
LIN {X 0,Y 128.676,Z 187.374,A -85,B 0,C 180,E1 -25533.086,E2 -25533.086} C_VEL
LIN {X 0,Y 127.082,Z 184.527,A -85,B 0,C 180,E1 -25535.168,E2 -25535.168} C_VEL
LIN {X 0,Y 126.262,Z 183.943,A -85,B 0,C 180,E1 -25536.199,E2 -25536.199} C_VEL
LIN {X 0,Y 123.509,Z 181.8,A -85,B 0,C 180,E1 -25540.253,E2 -25540.253} C_VEL
LIN {X 0,Y 122.258,Z 179.35,A -85,B 0,C 180,E1 -25542.865,E2 -25542.865} C_VEL
LIN {X 0,Y 122.064,Z 178.266,A -85,B 0,C 180,E1 -25543.591,E2 -25543.591} C_VEL
LIN {X 0,Y 122.382,Z 178.207,A -85,B 0,C 180,E1 -25550.079,E2 -25550.079} C_VEL
LIN {X 0,Y 122.545,Z 178.169,A -85,B 0,C 180,E1 -25556.712,E2 -25556.712} C_VEL
LIN {X 0,Y 123.011,Z 178.162,A -85,B 0,C 180,E1 -25560,E2 -25560} C_VEL
LIN {X 0,Y 122.396,Z 178.233,A -85,B 0,C 180,E1 -25566.594,E2 -25566.594} C_VEL
LIN {X 0,Y 122.34,Z 178.408,A -85,B 0,C 180,E1 -25571.464,E2 -25571.464} C_VEL
LIN {X 0,Y 123.038,Z 180.843,A -85,B 0,C 180,E1 -25573.207,E2 -25573.207} C_VEL
LIN {X 0,Y 125.024,Z 183.209,A -85,B 0,C 180,E1 -25576.533,E2 -25576.533} C_VEL
LIN {X 0,Y 127.216,Z 184.43,A -85,B 0,C 180,E1 -25579.358,E2 -25579.358} C_VEL
LIN {X 0,Y 128.65,Z 187.379,A -85,B 0,C 180,E1 -25581.281,E2 -25581.281} C_VEL
LIN {X 0,Y 131.117,Z 189.563,A -85,B 0,C 180,E1 -25583.861,E2 -25583.861} C_VEL
LIN {X 0,Y 134.088,Z 193.759,A -85,B 0,C 180,E1 -25586.745,E2 -25586.745} C_VEL
LIN {X 0,Y 135.391,Z 195.175,A -85,B 0,C 180,E1 -25587.851,E2 -25587.851} C_VEL
LIN {X 0,Y 138.158,Z 198.943,A -85,B 0,C 180,E1 -25590.096,E2 -25590.096} C_VEL
LIN {X 0,Y 142.291,Z 204.993,A -85,B 0,C 180,E1 -25593.107,E2 -25593.107} C_VEL
LIN {X 0,Y 145.537,Z 210.96,A -85,B 0,C 180,E1 -25595.313,E2 -25595.313} C_VEL
LIN {X 0,Y 150.613,Z 222.005,A -85,B 0,C 180,E1 -25598.51,E2 -25598.51} C_VEL
